REGION Network 28: pomocniczy bit ustawiania napędu dodatkowego nr2 / pomocniczy bit ustawiania pompy dodatkoweo nr2
   // Reset znacznika po udanym załączeniu pompy dodatkowej
   // Reset w wypadku braku pompy
   RUNG wire#powerrail
      I_Contact( "AlwaysTRUE" )
      wire#w1
      Contact( "Is_extras_K2_P1" )
      Contact( "IsRunNetwork_P1" )
      wire#w2
      R_Coil( #set_Motor3 )
   END_RUNG
   RUNG wire#w1
      Contact( "Is_extras_K2_P2" )
      Contact( "IsRunNetwork_P2" )
   END_RUNG wire#w2
   RUNG wire#w1
      Contact( "Is_extras_K2_P3" )
      Contact( "IsRunNetwork_P3" )
   END_RUNG wire#w2
   RUNG wire#w1
      Contact( "Is_extras_K2_P4" )
      Contact( "IsRunNetwork_P4" )
   END_RUNG wire#w2
   RUNG wire#w1
      Contact( "Reset_Motor3Alarm" )
   END_RUNG wire#w2
   RUNG wire#w1
      I_Contact( "IsModeAut" )
   END_RUNG wire#w2
   // the same network as SCL:
   IF NOT "AlwaysTRUE" AND (("Is_extras_K2_P1" AND "IsRunNetwork_P1") OR ("Is_extras_K2_P2" AND "IsRunNetwork_P2") OR ("Is_extras_K2_P3" AND "IsRunNetwork_P3") OR ("Is_extras_K2_P4" AND "IsRunNetwork_P4") OR "Reset_Motor3Alarm" OR NOT "IsModeAut") THEN
       #set_Motor3 := FALSE;
   END_IF;
END_REGION

REGION Network 29: pomocniczy bit ustawiania napędu dodatkowego nr2 / pomocniczy bit ustawiania pompy dodatkowe nr3
   // Reset znacznika po udanym załączeniu pompy dodatkowej
   // Reset w wypadku braku pompy
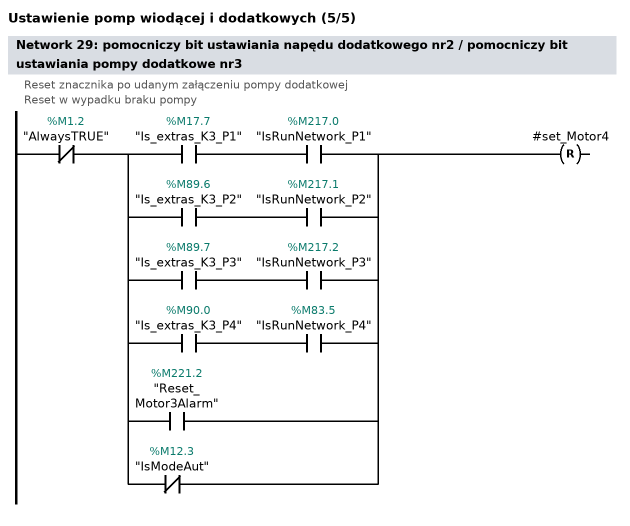
   RUNG wire#powerrail
      I_Contact( "AlwaysTRUE" )
      wire#w1
      Contact( "Is_extras_K3_P1" )
      Contact( "IsRunNetwork_P1" )
      wire#w2
      R_Coil( #set_Motor4 )
   END_RUNG
   RUNG wire#w1
      Contact( "Is_extras_K3_P2" )
      Contact( "IsRunNetwork_P2" )
   END_RUNG wire#w2
   RUNG wire#w1
      Contact( "Is_extras_K3_P3" )
      Contact( "IsRunNetwork_P3" )
   END_RUNG wire#w2
   RUNG wire#w1
      Contact( "Is_extras_K3_P4" )
      Contact( "IsRunNetwork_P4" )
   END_RUNG wire#w2
   RUNG wire#w1
      Contact( "Reset_Motor3Alarm" )
   END_RUNG wire#w2
   RUNG wire#w1
      I_Contact( "IsModeAut" )
   END_RUNG wire#w2
   // the same network as SCL:
   IF NOT "AlwaysTRUE" AND (("Is_extras_K3_P1" AND "IsRunNetwork_P1") OR ("Is_extras_K3_P2" AND "IsRunNetwork_P2") OR ("Is_extras_K3_P3" AND "IsRunNetwork_P3") OR ("Is_extras_K3_P4" AND "IsRunNetwork_P4") OR "Reset_Motor3Alarm" OR NOT "IsModeAut") THEN
       #set_Motor4 := FALSE;
   END_IF;
END_REGION
END_FUNCTION_BLOCK

FUNCTION_BLOCK "Sterowanie dołączeniem falownika"   // FB8, LAD
TITLE = Sterowanie dołączaniem styczników falownika
{ S7_Optimized_Access := 'TRUE' }
AUTHOR : rtecmer
VERSION : 0.1
// Sterowa stycznikiem pracy z falownika.
// Funkcja FB8 komutuje załaczenie stycznika FALOWNIK dla konkretnego napędu. Napędem sterowanym jest zawsze napęd przypisany do MC (czyli IsReady_MC to jest gotowość napędu sterowaniego) Na wejścia oznaczone wyróżnikiem MC podlączamy sygnały tej samej dmuchawy, której stycznikiem będziemy sterować poprzez wtjście setSUPV_FM
//  
// Sterowanie stycznikiem . Ustawianie znaczników setCMD_FM i setSUPV_FM które przekazywane są do funkcji FC3/FC1 DRV01 driver napędów. Następnie przekazywane jest do warstwy Hawtware/ OUT gdzie ustawiane jest wyjście sterownika
// stored: AutoNumber true, IsIECCheckEnabled false, IsRetainMemResEnabled false, MemoryReserve 500, SetENOAutomatically false, UDAEnableTagReadback false
   VAR_INPUT
      Is_up_Hz : Bool;
      Set_HWork_M : Bool;   // Znacznik ustawienia pracy od licznika
      setPID_Pompy : Bool;   // Znacznik załączenie, regulacji falownika
      IsRunInverter_MA : Bool;   // Potwierdzenie pracy z falownika kompresor dodatkowy 1
      IsRunNetwork_MA : Bool;   // Potwierdzenie praca z sieć dodatkowego
      IsRunInverter_MB : Bool;   // Potwierdzenie pracy z falownika kompresor dodatkowy 2
      IsRunNetwork_MB : Bool;   // Potwierdzenie praca z sieć dodatkowego
      IsRunNetwork_MC : Bool;   // Potwierdzenie pracy z sieci
      IsRunInverter_MC : Bool;   // Potwierdzenie pracy z falownika
      IsRunNetwork_MD : Bool;   // Potwierdzenie pracy z sieci
      IsRunInverter_MD : Bool;   // Potwierdzenie pracy z falownika
      FC2_Set_50H : Bool;   // Znacznik osiągnięcia czasu dla 50Hz
      IsRunInverter1 : Bool;   // Potwierdzenie pracy falownika / Potwierdzenie pracy falownika kompresorów M7M8M9
      AlwaysTRUE : Bool;
      IsReady_MA : Bool;   // Znacznik gotowości
      IsReady_MB : Bool;   // Znacznik gotowości
      IsReady_MC : Bool;   // Znacznik gotowości
      IsReady_MD : Bool;   // Znacznik gotowości
      IsModeAut : Bool;   // Znacznik trybu automat
      FB9_Set_Motor2 : Bool;   // Polecenie dostawienia dodatkowej nr1
      FB9_Set_Motor3 : Bool;   // Polecenie dostawienia dodatkowej nr2
      FB9_Set_Motor4 : Bool;   // Polecenie dostawienia dodatkowej nr3
      IsReady_Inverter : Bool;   // Gotowość falownika
      ResWorkInverter_to_MaxTime : Bool;   // Bit kasowania pracy falownika od maxymalnej ciągłej pracy
   END_VAR
   VAR_OUTPUT
      setSUPV_FM : Bool;   // Znacznik polecenia startu z falownika
   END_VAR
   VAR_IN_OUT
      setCMD_FM : Bool;   // Znacznik sterowania w trybie falownik
      Timer_OFF_Inverter_M : TOF_TIME;   // Timer na blokowanie po odłączeniu stycznika falownika
      Timer_Start_Inver_M : TON_TIME;   // Timer opóźnienia załaczenia stycznika pracy z falownika
      Timer_Set50Hz_Off_Inver_M : TON_TIME;   // Timer opóźnieniawyłączeniea falownika
      Mem_Res_setCMD_MC : Bool;   // pamięć zbocza załączenia timera blokowania stycznika falowni
   END_VAR
   VAR
      Network_50Hz : Bool;   // Znacznik 50 Hz podtrzymanie przełączenia na sieć
   END_VAR
   VAR_TEMP
      IsDrive_Optimum : Bool;   // Znacznik optymalnej ilości napędów. Jeśli False to nie przełaczaj Falowni/Sieć
      CMD_OFF_inverter : Bool;   // Wyłączenie falownika od 50Hz i dodatkowa / Wyłączenie falownika od 50Hz i udtawiona dodatkowa
      tmpOFF_inverter : Bool;
   END_VAR
   VAR_TEMP   // added for the SCL form of the ladder/FBD networks
      _w1 : Bool;
      _w2 : Bool;
   END_VAR
BEGIN

REGION Network 1: Control status motors / Kontrola statusu napędu
   // // Dostępna  jedna dmuchawa gdy wartość 1, 2, 4
   // // Dostępne dwie dmuchawy gdy wartość 6, 5, 3 
   // // Dostępne trzy dmuchawy gdy wartość 7
END_REGION

REGION Network 2: Histereza na dołączenie stycznika falownika
   // Sterowanie dołączeniem stycznika pracy z falownika
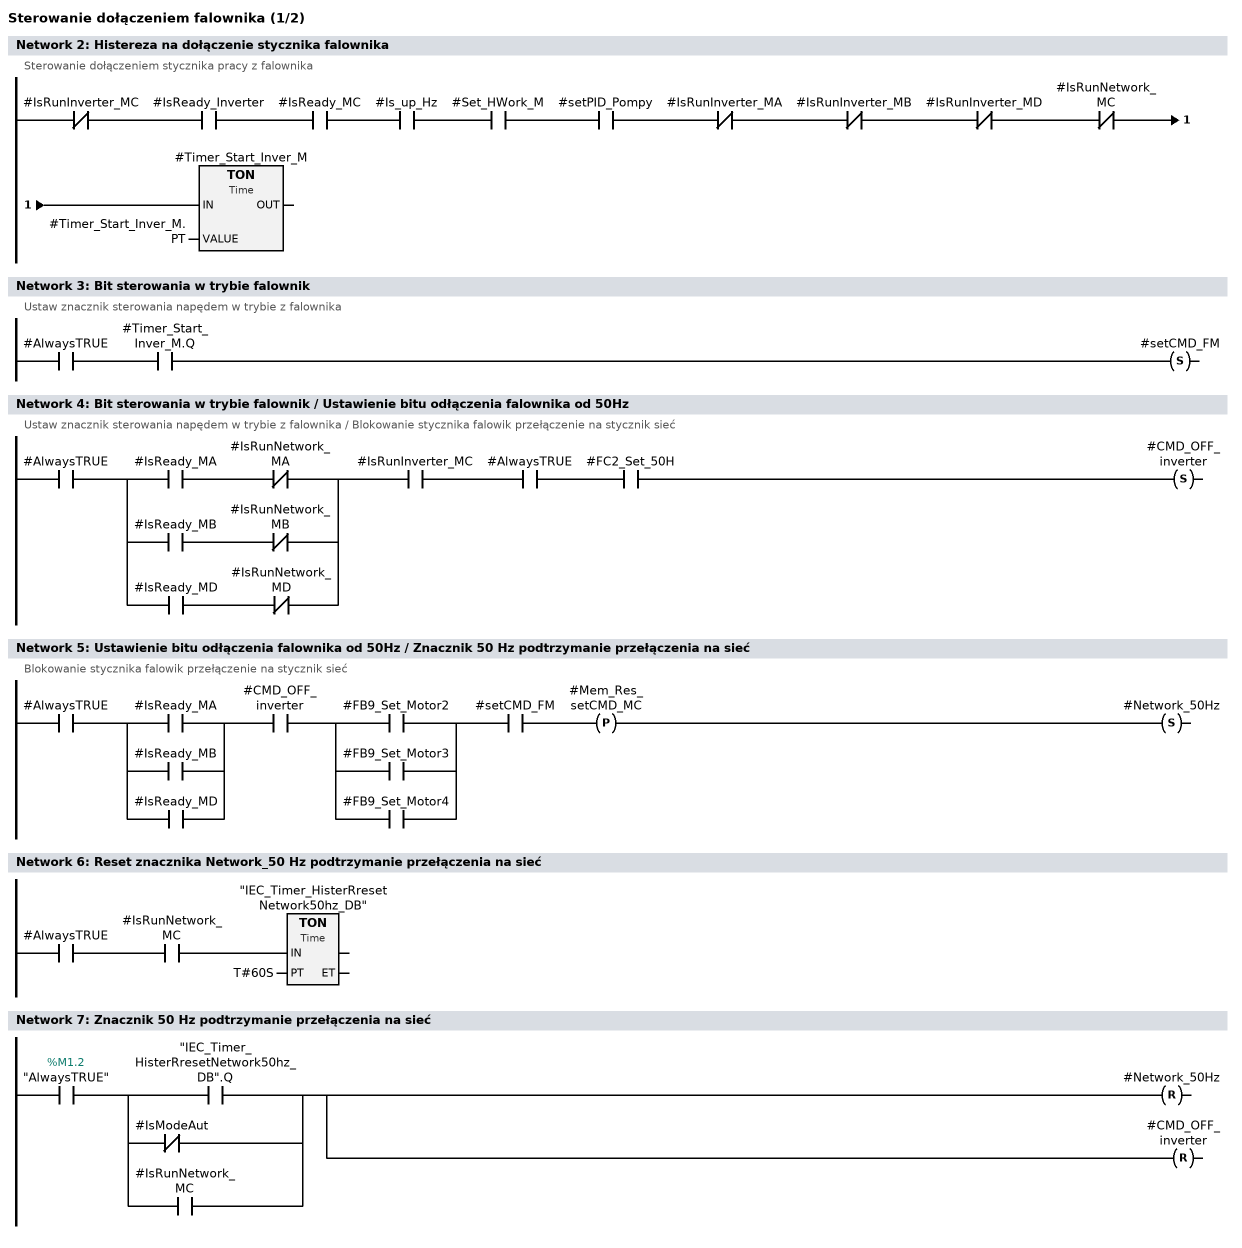
   #Timer_Start_Inver_M(IN := NOT #IsRunInverter_MC AND #IsReady_Inverter AND #IsReady_MC AND #Is_up_Hz AND #Set_HWork_M AND #setPID_Pompy AND NOT #IsRunInverter_MA AND NOT #IsRunInverter_MB AND NOT #IsRunInverter_MD AND NOT #IsRunNetwork_MC, PT := #Timer_Start_Inver_M.PT);   // TON coil
END_REGION

REGION Network 3: Bit sterowania w trybie falownik
   // Ustaw znacznik sterowania napędem w trybie z falownika
   RUNG wire#powerrail
      Contact( #AlwaysTRUE )
      Contact( #Timer_Start_Inver_M.Q )
      S_Coil( #setCMD_FM )
   END_RUNG
   // the same network as SCL:
   IF #AlwaysTRUE AND #Timer_Start_Inver_M.Q THEN #setCMD_FM := TRUE; END_IF;
END_REGION

REGION Network 4: Bit sterowania w trybie falownik / Ustawienie bitu odłączenia falownika od 50Hz
   // Ustaw znacznik sterowania napędem w trybie z falownika / Blokowanie stycznika falowik przełączenie na stycznik sieć
   RUNG wire#powerrail
      Contact( #AlwaysTRUE )
      wire#w1
      Contact( #IsReady_MA )
      I_Contact( #IsRunNetwork_MA )
      wire#w2
      Contact( #IsRunInverter_MC )
      Contact( #AlwaysTRUE )
      Contact( #FC2_Set_50H )
      S_Coil( #CMD_OFF_inverter )
   END_RUNG
   RUNG wire#w1
      Contact( #IsReady_MB )
      I_Contact( #IsRunNetwork_MB )
   END_RUNG wire#w2
   RUNG wire#w1
      Contact( #IsReady_MD )
      I_Contact( #IsRunNetwork_MD )
   END_RUNG wire#w2
   // the same network as SCL:
   IF #AlwaysTRUE AND ((#IsReady_MA AND NOT #IsRunNetwork_MA) OR (#IsReady_MB AND NOT #IsRunNetwork_MB) OR (#IsReady_MD AND NOT #IsRunNetwork_MD)) AND #IsRunInverter_MC AND #AlwaysTRUE AND #FC2_Set_50H THEN
       #CMD_OFF_inverter := TRUE;
   END_IF;
END_REGION

REGION Network 5: Ustawienie bitu odłączenia falownika od 50Hz / Znacznik 50 Hz podtrzymanie przełączenia na sieć
   // Blokowanie stycznika falowik przełączenie na stycznik sieć
   RUNG wire#powerrail
      Contact( #AlwaysTRUE )
      wire#w1
      Contact( #IsReady_MA )
      wire#w2
      Contact( #CMD_OFF_inverter )
      wire#w3
      Contact( #FB9_Set_Motor2 )
      wire#w4
      Contact( #setCMD_FM )
      P_Trig( #Mem_Res_setCMD_MC )
      S_Coil( #Network_50Hz )
   END_RUNG
   RUNG wire#w1
      Contact( #IsReady_MB )
   END_RUNG wire#w2
   RUNG wire#w1
      Contact( #IsReady_MD )
   END_RUNG wire#w2
   RUNG wire#w3
      Contact( #FB9_Set_Motor3 )
   END_RUNG wire#w4
   RUNG wire#w3
      Contact( #FB9_Set_Motor4 )
   END_RUNG wire#w4
   // the same network as SCL:
   #_w1 := #AlwaysTRUE AND (#IsReady_MA OR #IsReady_MB OR #IsReady_MD) AND #CMD_OFF_inverter AND (#FB9_Set_Motor2 OR #FB9_Set_Motor3 OR #FB9_Set_Motor4) AND #setCMD_FM;
   #_w2 := #_w1 AND NOT #Mem_Res_setCMD_MC;   // rising edge
   #Mem_Res_setCMD_MC := #_w1;
   IF #_w2 THEN #Network_50Hz := TRUE; END_IF;
END_REGION

REGION Network 6: Reset znacznika Network_50 Hz podtrzymanie przełączenia na sieć
   RUNG wire#powerrail
      Contact( #AlwaysTRUE )
      Contact( #IsRunNetwork_MC )
      { S7_Templates := "time_type := Time" } "IEC_Timer_HisterRresetNetwork50hz_DB".TON(pt := T#60S, et =>)
   END_RUNG
   // the same network as SCL:
   "IEC_Timer_HisterRresetNetwork50hz_DB".TON(IN := #AlwaysTRUE AND #IsRunNetwork_MC, PT := T#60S);
END_REGION

REGION Network 7: Znacznik 50 Hz podtrzymanie przełączenia na sieć
   RUNG wire#powerrail
      Contact( "AlwaysTRUE" )
      wire#w1
      Contact( "IEC_Timer_HisterRresetNetwork50hz_DB".Q )
      wire#w2
      R_Coil( #Network_50Hz )
   END_RUNG
   RUNG wire#w1
      I_Contact( #IsModeAut )
   END_RUNG wire#w2
   RUNG wire#w1
      Contact( #IsRunNetwork_MC )
   END_RUNG wire#w2
   RUNG wire#w2
      R_Coil( #CMD_OFF_inverter )
   END_RUNG
   // the same network as SCL:
   IF "AlwaysTRUE" AND ("IEC_Timer_HisterRresetNetwork50hz_DB".Q OR NOT #IsModeAut OR #IsRunNetwork_MC) THEN
       #Network_50Hz := FALSE;
       #CMD_OFF_inverter := FALSE;
   END_IF;
END_REGION

REGION Network 8: Timer blokowania po odłączenieu stycznika falownik
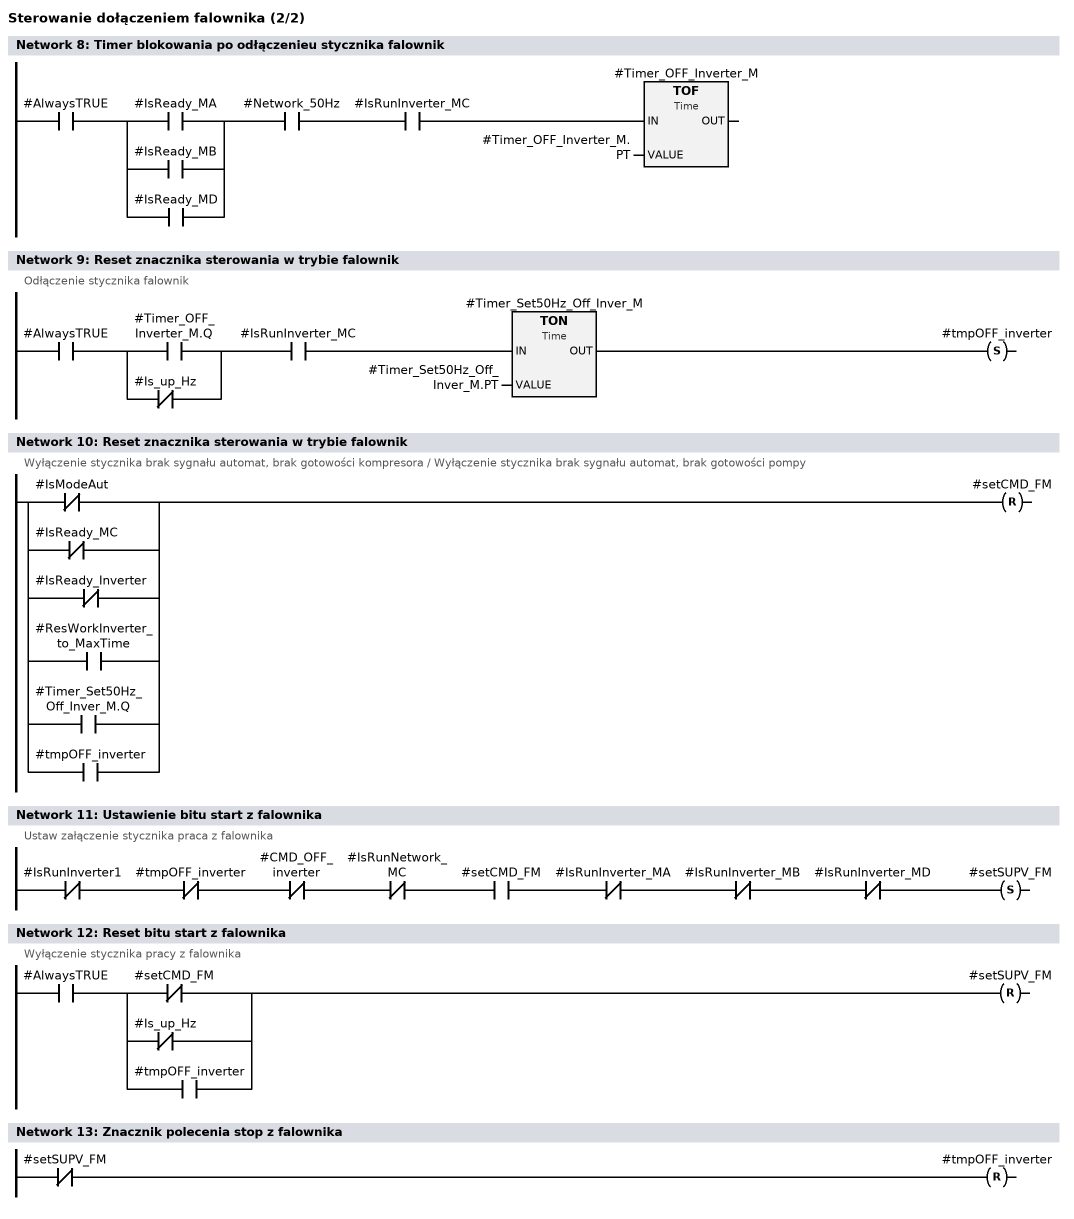
   #Timer_OFF_Inverter_M(IN := #AlwaysTRUE AND (#IsReady_MA OR #IsReady_MB OR #IsReady_MD) AND #Network_50Hz AND #IsRunInverter_MC, PT := #Timer_OFF_Inverter_M.PT);   // TOF coil
END_REGION

REGION Network 9: Reset znacznika sterowania w trybie falownik
   // Odłączenie stycznika falownik
   #_w1 := #AlwaysTRUE AND (#Timer_OFF_Inverter_M.Q OR NOT #Is_up_Hz) AND #IsRunInverter_MC;
   #Timer_Set50Hz_Off_Inver_M(IN := #_w1, PT := #Timer_Set50Hz_Off_Inver_M.PT);   // TON coil
   IF #_w1 THEN #tmpOFF_inverter := TRUE; END_IF;
END_REGION

REGION Network 10: Reset znacznika sterowania w trybie falownik
   // Wyłączenie stycznika brak sygnału automat, brak gotowości kompresora / Wyłączenie stycznika brak sygnału automat, brak gotowości pompy
   RUNG wire#powerrail
      I_Contact( #IsModeAut )
      wire#w1
      R_Coil( #setCMD_FM )
   END_RUNG
   RUNG wire#powerrail
      I_Contact( #IsReady_MC )
   END_RUNG wire#w1
   RUNG wire#powerrail
      I_Contact( #IsReady_Inverter )
   END_RUNG wire#w1
   RUNG wire#powerrail
      Contact( #ResWorkInverter_to_MaxTime )
   END_RUNG wire#w1
   RUNG wire#powerrail
      Contact( #Timer_Set50Hz_Off_Inver_M.Q )
   END_RUNG wire#w1
   RUNG wire#powerrail
      Contact( #tmpOFF_inverter )
   END_RUNG wire#w1
   // the same network as SCL:
   IF NOT #IsModeAut OR NOT #IsReady_MC OR NOT #IsReady_Inverter OR #ResWorkInverter_to_MaxTime OR #Timer_Set50Hz_Off_Inver_M.Q OR #tmpOFF_inverter THEN
       #setCMD_FM := FALSE;
   END_IF;
END_REGION

REGION Network 11: Ustawienie bitu start z falownika
   // Ustaw załączenie stycznika praca z falownika
   RUNG wire#powerrail
      I_Contact( #IsRunInverter1 )
      I_Contact( #tmpOFF_inverter )
      I_Contact( #CMD_OFF_inverter )
      I_Contact( #IsRunNetwork_MC )
      Contact( #setCMD_FM )
      I_Contact( #IsRunInverter_MA )
      I_Contact( #IsRunInverter_MB )
      I_Contact( #IsRunInverter_MD )
      S_Coil( #setSUPV_FM )
   END_RUNG
   // the same network as SCL:
   IF NOT #IsRunInverter1 AND NOT #tmpOFF_inverter AND NOT #CMD_OFF_inverter AND NOT #IsRunNetwork_MC AND #setCMD_FM AND NOT #IsRunInverter_MA AND NOT #IsRunInverter_MB AND NOT #IsRunInverter_MD THEN
       #setSUPV_FM := TRUE;
   END_IF;
END_REGION

REGION Network 12: Reset bitu start z falownika
   // Wyłączenie stycznika pracy z falownika
   RUNG wire#powerrail
      Contact( #AlwaysTRUE )
      wire#w1
      I_Contact( #setCMD_FM )
      wire#w2
      R_Coil( #setSUPV_FM )
   END_RUNG
   RUNG wire#w1
      I_Contact( #Is_up_Hz )
   END_RUNG wire#w2
   RUNG wire#w1
      Contact( #tmpOFF_inverter )
   END_RUNG wire#w2
   // the same network as SCL:
   IF #AlwaysTRUE AND (NOT #setCMD_FM OR NOT #Is_up_Hz OR #tmpOFF_inverter) THEN
       #setSUPV_FM := FALSE;
   END_IF;
END_REGION

REGION Network 13: Znacznik polecenia stop z falownika
   RUNG wire#powerrail
      I_Contact( #setSUPV_FM )
      R_Coil( #tmpOFF_inverter )
   END_RUNG
   // the same network as SCL:
   IF NOT #setSUPV_FM THEN #tmpOFF_inverter := FALSE; END_IF;
END_REGION
END_FUNCTION_BLOCK

FUNCTION "Korekta Tryb Pracy" : Void   // FC34, LAD
TITLE = potrzymanie trybu
{ S7_Optimized_Access := 'TRUE' }
AUTHOR : rtecmer
VERSION : 0.1
// z powodu P1 dodanyblok potzymujący tryb pracy napędów podczas przełączania falowni / siec
// stored: AutoNumber true, IsIECCheckEnabled false, SetENOAutomatically false, UDAEnableTagReadback false
   VAR_TEMP   // added for the SCL form of the ladder/FBD networks
      _w1 : Bool;
   END_VAR
BEGIN

REGION Network 2: Ustawienie pracy [Automat]
   // Ustawienie bitu [Automat] przełacznikiem trybu pracy
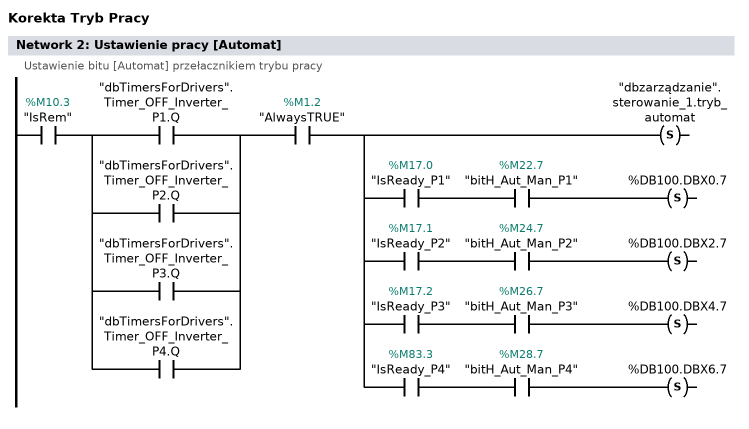
   RUNG wire#powerrail
      Contact( "IsRem" )
      wire#w1
      Contact( "dbTimersForDrivers".Timer_OFF_Inverter_P1.Q )
      wire#w2
      Contact( "AlwaysTRUE" )
      wire#w3
      S_Coil( "dbzarządzanie".sterowanie_1.tryb_automat )
   END_RUNG
   RUNG wire#w1
      Contact( "dbTimersForDrivers".Timer_OFF_Inverter_P2.Q )
   END_RUNG wire#w2
   RUNG wire#w1
      Contact( "dbTimersForDrivers".Timer_OFF_Inverter_P3.Q )
   END_RUNG wire#w2
   RUNG wire#w1
      Contact( "dbTimersForDrivers".Timer_OFF_Inverter_P4.Q )
   END_RUNG wire#w2
   RUNG wire#w3
      Contact( "IsReady_P1" )
      Contact( "bitH_Aut_Man_P1" )
      S_Coil( %DB100.DBX0.7 )
   END_RUNG
   RUNG wire#w3
      Contact( "IsReady_P2" )
      Contact( "bitH_Aut_Man_P2" )
      S_Coil( %DB100.DBX2.7 )
   END_RUNG
   RUNG wire#w3
      Contact( "IsReady_P3" )
      Contact( "bitH_Aut_Man_P3" )
      S_Coil( %DB100.DBX4.7 )
   END_RUNG
   RUNG wire#w3
      Contact( "IsReady_P4" )
      Contact( "bitH_Aut_Man_P4" )
      S_Coil( %DB100.DBX6.7 )
   END_RUNG
   // the same network as SCL:
   #_w1 := "IsRem" AND ("dbTimersForDrivers".Timer_OFF_Inverter_P1.Q OR "dbTimersForDrivers".Timer_OFF_Inverter_P2.Q OR "dbTimersForDrivers".Timer_OFF_Inverter_P3.Q OR "dbTimersForDrivers".Timer_OFF_Inverter_P4.Q) AND "AlwaysTRUE";
   IF #_w1 THEN "dbzarządzanie".sterowanie_1.tryb_automat := TRUE; END_IF;
   IF #_w1 AND "IsReady_P1" AND "bitH_Aut_Man_P1" THEN %DB100.DBX0.7 := TRUE; END_IF;
   IF #_w1 AND "IsReady_P2" AND "bitH_Aut_Man_P2" THEN %DB100.DBX2.7 := TRUE; END_IF;
   IF #_w1 AND "IsReady_P3" AND "bitH_Aut_Man_P3" THEN %DB100.DBX4.7 := TRUE; END_IF;
   IF #_w1 AND "IsReady_P4" AND "bitH_Aut_Man_P4" THEN %DB100.DBX6.7 := TRUE; END_IF;
END_REGION
END_FUNCTION

FUNCTION_BLOCK "Sterowanie falownikiem"   // FB11, LAD
TITLE = Control of Inverters
{ S7_Optimized_Access := 'TRUE' }
AUTHOR : rtecmer
VERSION : 0.1
// Sterowanie przekaćnikiem załączającym falownik do pracy
// stored: AutoNumber true, IsIECCheckEnabled false, IsRetainMemResEnabled false, MemoryReserve 500, SetENOAutomatically false, UDAEnableTagReadback false
   VAR_INPUT
      IsModeAut : Bool;   // Znacznik tryb automat dla pomp
      AlwaysTRUE : Bool;
      Set_HWork_P1 : Bool;   // Znacznik ustawienia pracy od licznika pracy
      Set_HWork_P2 : Bool;   // Znacznik ustawienia pracy od licznika pracy
      Set_HWork_P3 : Bool;   // Znacznik ustawienia pracy od licznika pracy
      Set_HWork_P4 : Bool;
      setPID_Pomp : Bool;   // Znacznik załączenie, regulacji falownika
      Is_loading_K3 : Bool;   // Znacznik pompy wiodącej
      IsRunInverter_P4 : Bool;
      IsRunInverter_P3 : Bool;   // Potwierdzenie załączenie stycznika falownik pompy
      IsRunInverter_P2 : Bool;   // Potwierdzenie załączenie stycznika falownik pompy
      IsRunInverter_P1 : Bool;   // Potwierdzenie załączenie stycznika falownik pompy
      Bit_Aut_P1 : Bool;   // Bit tryb prac automat
      Bit_Aut_P2 : Bool;   // Bit tryb prac automat
      Bit_Aut_P3 : Bool;   // Bit tryb prac automat
      Bit_Aut_P4 : Bool;
      IsRunNetwork_P1 : Bool;   // Potwierdzenie załączenie stycznika sieć
      IsRunNetwork_P2 : Bool := false;   // Potwierdzenie załączenie stycznika sieć
      IsRunNetwork_P3 : Bool := false;   // Potwierdzenie załączenie stycznika sieć
      IsRunNetwork_P4 : Bool;
   END_VAR
   VAR_OUTPUT
      CMD_start_stop_inverter : Bool;   // Przekaźnik sterowania załączaniem falownika
   END_VAR
   VAR
      Res_upHz : Bool;   // Reset znacznika up_Hz wyłaczenie dodatkowe
   END_VAR
BEGIN

REGION Network 1: Reset bitu pomocniczego ustalenia przyrostu Hz
   // Kasowanie podczas rozruchu po restarcie
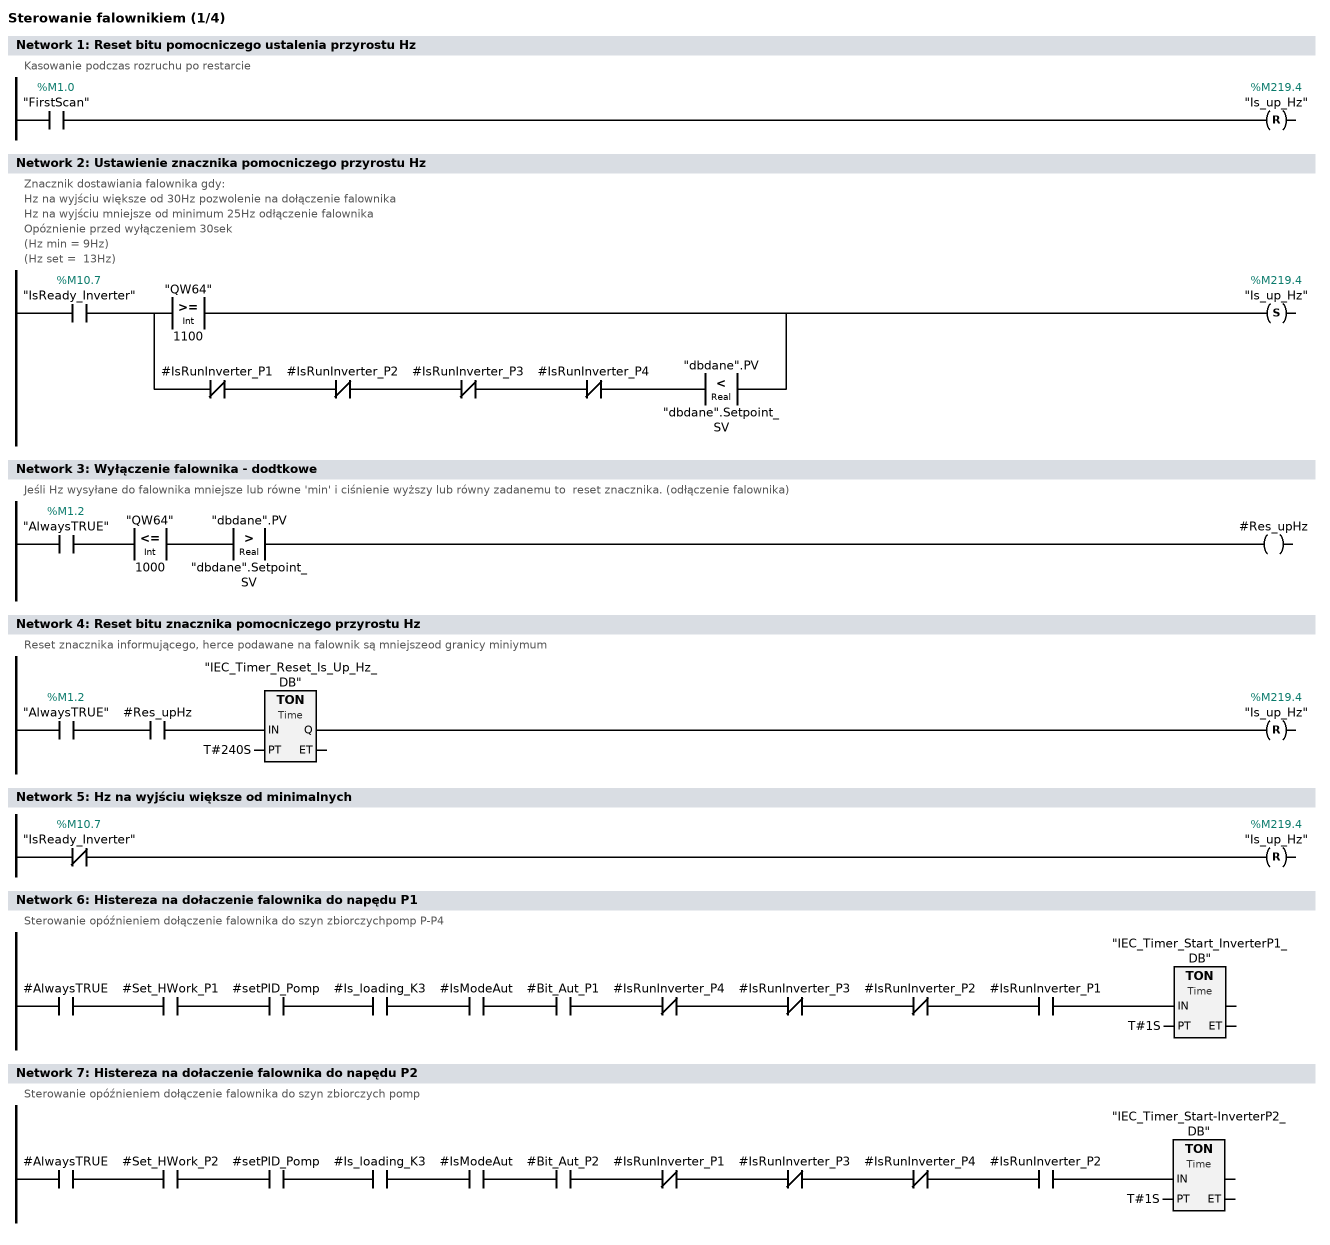
   RUNG wire#powerrail
      Contact( "FirstScan" )
      R_Coil( "Is_up_Hz" )
   END_RUNG
   // the same network as SCL:
   IF "FirstScan" THEN "Is_up_Hz" := FALSE; END_IF;
END_REGION

REGION Network 2: Ustawienie znacznika pomocniczego przyrostu Hz
   // Znacznik dostawiania falownika gdy:
   // Hz na wyjściu większe od 30Hz pozwolenie na dołączenie falownika
   // Hz na wyjściu mniejsze od minimum 25Hz odłączenie falownika
   // Opóznienie przed wyłączeniem 30sek
   // (Hz min = 9Hz)
   // (Hz set =  13Hz)
   RUNG wire#powerrail
      Contact( "IsReady_Inverter" )
      wire#w1
      { S7_Templates := "SrcType := Int" } GE_Contact(in1 := "QW64", in2 := 1100)
      wire#w2
      S_Coil( "Is_up_Hz" )
   END_RUNG
   RUNG wire#w1
      I_Contact( #IsRunInverter_P1 )
      I_Contact( #IsRunInverter_P2 )
      I_Contact( #IsRunInverter_P3 )
      I_Contact( #IsRunInverter_P4 )
      { S7_Templates := "SrcType := Real" } LT_Contact(in1 := "dbdane".PV, in2 := "dbdane".Setpoint_SV)
   END_RUNG wire#w2
   // the same network as SCL:
   IF "IsReady_Inverter" AND (("QW64" >= 1100) OR (NOT #IsRunInverter_P1 AND NOT #IsRunInverter_P2 AND NOT #IsRunInverter_P3 AND NOT #IsRunInverter_P4 AND ("dbdane".PV < "dbdane".Setpoint_SV))) THEN
       "Is_up_Hz" := TRUE;
   END_IF;
END_REGION

REGION Network 3: Wyłączenie falownika - dodtkowe
   // Jeśli Hz wysyłane do falownika mniejsze lub równe 'min' i ciśnienie wyższy lub równy zadanemu to  reset znacznika. (odłączenie falownika)
   RUNG wire#powerrail
      Contact( "AlwaysTRUE" )
      { S7_Templates := "SrcType := Int" } LE_Contact(in1 := "QW64", in2 := 1000)
      { S7_Templates := "SrcType := Real" } GT_Contact(in1 := "dbdane".PV, in2 := "dbdane".Setpoint_SV)
      Coil( #Res_upHz )
   END_RUNG
   // the same network as SCL:
   #Res_upHz := "AlwaysTRUE" AND ("QW64" <= 1000) AND ("dbdane".PV > "dbdane".Setpoint_SV);
END_REGION

REGION Network 4: Reset bitu znacznika pomocniczego przyrostu Hz
   // Reset znacznika informującego, herce podawane na falownik są mniejszeod granicy miniymum
   RUNG wire#powerrail
      Contact( "AlwaysTRUE" )
      Contact( #Res_upHz )
      { S7_Templates := "time_type := Time" } "IEC_Timer_Reset_Is_Up_Hz_DB".TON(pt := T#240S, et =>)
      R_Coil( "Is_up_Hz" )
   END_RUNG
   // the same network as SCL:
   "IEC_Timer_Reset_Is_Up_Hz_DB".TON(IN := "AlwaysTRUE" AND #Res_upHz, PT := T#240S);
   IF "IEC_Timer_Reset_Is_Up_Hz_DB".Q THEN "Is_up_Hz" := FALSE; END_IF;
END_REGION

REGION Network 5: Hz na wyjściu większe od minimalnych
   RUNG wire#powerrail
      I_Contact( "IsReady_Inverter" )
      R_Coil( "Is_up_Hz" )
   END_RUNG
   // the same network as SCL:
   IF NOT "IsReady_Inverter" THEN "Is_up_Hz" := FALSE; END_IF;
END_REGION

REGION Network 6: Histereza na dołaczenie falownika do napędu P1
   // Sterowanie opóźnieniem dołączenie falownika do szyn zbiorczychpomp P-P4
   RUNG wire#powerrail
      Contact( #AlwaysTRUE )
      Contact( #Set_HWork_P1 )
      Contact( #setPID_Pomp )
      Contact( #Is_loading_K3 )
      Contact( #IsModeAut )
      Contact( #Bit_Aut_P1 )
      I_Contact( #IsRunInverter_P4 )
      I_Contact( #IsRunInverter_P3 )
      I_Contact( #IsRunInverter_P2 )
      Contact( #IsRunInverter_P1 )
      { S7_Templates := "time_type := Time" } "IEC_Timer_Start_InverterP1_DB".TON(pt := T#1S, et =>)
   END_RUNG
   // the same network as SCL:
   "IEC_Timer_Start_InverterP1_DB".TON(IN := #AlwaysTRUE AND #Set_HWork_P1 AND #setPID_Pomp AND #Is_loading_K3 AND #IsModeAut AND #Bit_Aut_P1 AND NOT #IsRunInverter_P4 AND NOT #IsRunInverter_P3 AND NOT #IsRunInverter_P2 AND #IsRunInverter_P1,
                           PT := T#1S);
END_REGION

REGION Network 7: Histereza na dołaczenie falownika do napędu P2
   // Sterowanie opóźnieniem dołączenie falownika do szyn zbiorczych pomp
   RUNG wire#powerrail
      Contact( #AlwaysTRUE )
      Contact( #Set_HWork_P2 )
      Contact( #setPID_Pomp )
      Contact( #Is_loading_K3 )
      Contact( #IsModeAut )
      Contact( #Bit_Aut_P2 )
      I_Contact( #IsRunInverter_P1 )
      I_Contact( #IsRunInverter_P3 )
      I_Contact( #IsRunInverter_P4 )
      Contact( #IsRunInverter_P2 )
      { S7_Templates := "time_type := Time" } "IEC_Timer_Start-InverterP2_DB".TON(pt := T#1S, et =>)
   END_RUNG
   // the same network as SCL:
   "IEC_Timer_Start-InverterP2_DB".TON(IN := #AlwaysTRUE AND #Set_HWork_P2 AND #setPID_Pomp AND #Is_loading_K3 AND #IsModeAut AND #Bit_Aut_P2 AND NOT #IsRunInverter_P1 AND NOT #IsRunInverter_P3 AND NOT #IsRunInverter_P4 AND #IsRunInverter_P2,
                           PT := T#1S);
END_REGION

REGION Network 8: Histereza na dołaczenie falownika do napędu P3
   // Sterowanie opóźnieniem dołączenie falownika do szyn zbiorczych kompresorów
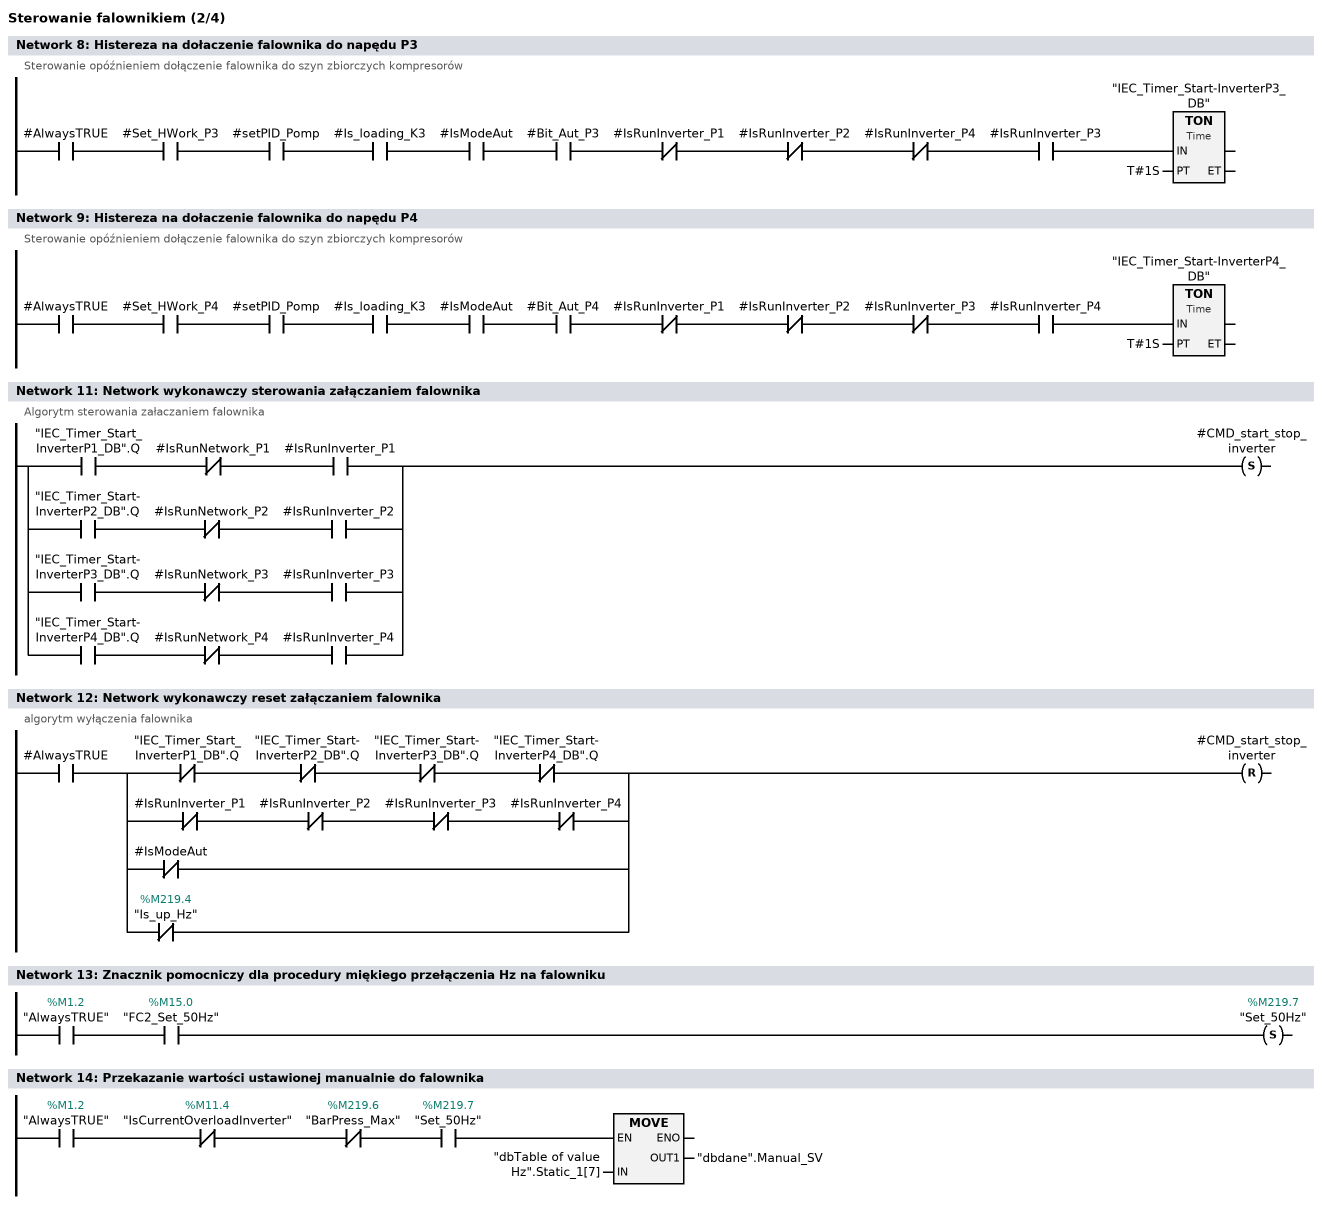
   RUNG wire#powerrail
      Contact( #AlwaysTRUE )
      Contact( #Set_HWork_P3 )
      Contact( #setPID_Pomp )
      Contact( #Is_loading_K3 )
      Contact( #IsModeAut )
      Contact( #Bit_Aut_P3 )
      I_Contact( #IsRunInverter_P1 )
      I_Contact( #IsRunInverter_P2 )
      I_Contact( #IsRunInverter_P4 )
      Contact( #IsRunInverter_P3 )
      { S7_Templates := "time_type := Time" } "IEC_Timer_Start-InverterP3_DB".TON(pt := T#1S, et =>)
   END_RUNG
   // the same network as SCL:
   "IEC_Timer_Start-InverterP3_DB".TON(IN := #AlwaysTRUE AND #Set_HWork_P3 AND #setPID_Pomp AND #Is_loading_K3 AND #IsModeAut AND #Bit_Aut_P3 AND NOT #IsRunInverter_P1 AND NOT #IsRunInverter_P2 AND NOT #IsRunInverter_P4 AND #IsRunInverter_P3,
                           PT := T#1S);
END_REGION

REGION Network 9: Histereza na dołaczenie falownika do napędu P4
   // Sterowanie opóźnieniem dołączenie falownika do szyn zbiorczych kompresorów
   RUNG wire#powerrail
      Contact( #AlwaysTRUE )
      Contact( #Set_HWork_P4 )
      Contact( #setPID_Pomp )
      Contact( #Is_loading_K3 )
      Contact( #IsModeAut )
      Contact( #Bit_Aut_P4 )
      I_Contact( #IsRunInverter_P1 )
      I_Contact( #IsRunInverter_P2 )
      I_Contact( #IsRunInverter_P3 )
      Contact( #IsRunInverter_P4 )
      { S7_Templates := "time_type := Time" } "IEC_Timer_Start-InverterP4_DB".TON(pt := T#1S, et =>)
   END_RUNG
   // the same network as SCL:
   "IEC_Timer_Start-InverterP4_DB".TON(IN := #AlwaysTRUE AND #Set_HWork_P4 AND #setPID_Pomp AND #Is_loading_K3 AND #IsModeAut AND #Bit_Aut_P4 AND NOT #IsRunInverter_P1 AND NOT #IsRunInverter_P2 AND NOT #IsRunInverter_P3 AND #IsRunInverter_P4,
                           PT := T#1S);
END_REGION

REGION Network 11: Network wykonawczy sterowania załączaniem falownika
   // Algorytm sterowania załaczaniem falownika
   RUNG wire#powerrail
      Contact( "IEC_Timer_Start_InverterP1_DB".Q )
      I_Contact( #IsRunNetwork_P1 )
      Contact( #IsRunInverter_P1 )
      wire#w1
      S_Coil( #CMD_start_stop_inverter )
   END_RUNG
   RUNG wire#powerrail
      Contact( "IEC_Timer_Start-InverterP2_DB".Q )
      I_Contact( #IsRunNetwork_P2 )
      Contact( #IsRunInverter_P2 )
   END_RUNG wire#w1
   RUNG wire#powerrail
      Contact( "IEC_Timer_Start-InverterP3_DB".Q )
      I_Contact( #IsRunNetwork_P3 )
      Contact( #IsRunInverter_P3 )
   END_RUNG wire#w1
   RUNG wire#powerrail
      Contact( "IEC_Timer_Start-InverterP4_DB".Q )
      I_Contact( #IsRunNetwork_P4 )
      Contact( #IsRunInverter_P4 )
   END_RUNG wire#w1
   // the same network as SCL:
   IF ("IEC_Timer_Start_InverterP1_DB".Q AND NOT #IsRunNetwork_P1 AND #IsRunInverter_P1) OR ("IEC_Timer_Start-InverterP2_DB".Q AND NOT #IsRunNetwork_P2 AND #IsRunInverter_P2) OR ("IEC_Timer_Start-InverterP3_DB".Q AND NOT #IsRunNetwork_P3 AND #IsRunInverter_P3) OR ("IEC_Timer_Start-InverterP4_DB".Q AND NOT #IsRunNetwork_P4 AND #IsRunInverter_P4) THEN
       #CMD_start_stop_inverter := TRUE;
   END_IF;
END_REGION

REGION Network 12: Network wykonawczy reset załączaniem falownika
   // algorytm wyłączenia falownika
   RUNG wire#powerrail
      Contact( #AlwaysTRUE )
      wire#w1
      I_Contact( "IEC_Timer_Start_InverterP1_DB".Q )
      I_Contact( "IEC_Timer_Start-InverterP2_DB".Q )
      I_Contact( "IEC_Timer_Start-InverterP3_DB".Q )
      I_Contact( "IEC_Timer_Start-InverterP4_DB".Q )
      wire#w2
      R_Coil( #CMD_start_stop_inverter )
   END_RUNG
   RUNG wire#w1
      I_Contact( #IsRunInverter_P1 )
      I_Contact( #IsRunInverter_P2 )
      I_Contact( #IsRunInverter_P3 )
      I_Contact( #IsRunInverter_P4 )
   END_RUNG wire#w2
   RUNG wire#w1
      I_Contact( #IsModeAut )
   END_RUNG wire#w2
   RUNG wire#w1
      I_Contact( "Is_up_Hz" )
   END_RUNG wire#w2
   // the same network as SCL:
   IF #AlwaysTRUE AND ((NOT "IEC_Timer_Start_InverterP1_DB".Q AND NOT "IEC_Timer_Start-InverterP2_DB".Q AND NOT "IEC_Timer_Start-InverterP3_DB".Q AND NOT "IEC_Timer_Start-InverterP4_DB".Q) OR (NOT #IsRunInverter_P1 AND NOT #IsRunInverter_P2 AND NOT #IsRunInverter_P3 AND NOT #IsRunInverter_P4) OR NOT #IsModeAut OR NOT "Is_up_Hz") THEN
       #CMD_start_stop_inverter := FALSE;
   END_IF;
END_REGION

REGION Network 13: Znacznik pomocniczy dla procedury miękiego przełączenia Hz na falowniku
   RUNG wire#powerrail
      Contact( "AlwaysTRUE" )
      Contact( "FC2_Set_50Hz" )
      S_Coil( "Set_50Hz" )
   END_RUNG
   // the same network as SCL:
   IF "AlwaysTRUE" AND "FC2_Set_50Hz" THEN "Set_50Hz" := TRUE; END_IF;
END_REGION

REGION Network 14: Przekazanie wartości ustawionej manualnie do falownika
   RUNG wire#powerrail
      Contact( "AlwaysTRUE" )
      I_Contact( "IsCurrentOverloadInverter" )
      I_Contact( "BarPress_Max" )
      Contact( "Set_50Hz" )
      Move(in := "dbTable of value Hz".Static_1[7], out1 => "dbdane".Manual_SV)
   END_RUNG
   // the same network as SCL:
   IF "AlwaysTRUE" AND NOT "IsCurrentOverloadInverter" AND NOT "BarPress_Max" AND "Set_50Hz" THEN
       "dbdane".Manual_SV := "dbTable of value Hz".Static_1[7];
   END_IF;
END_REGION

REGION Network 15: Przekazanie wartości ustawionej manualnie do falownika gdy awaria max ciśnienie
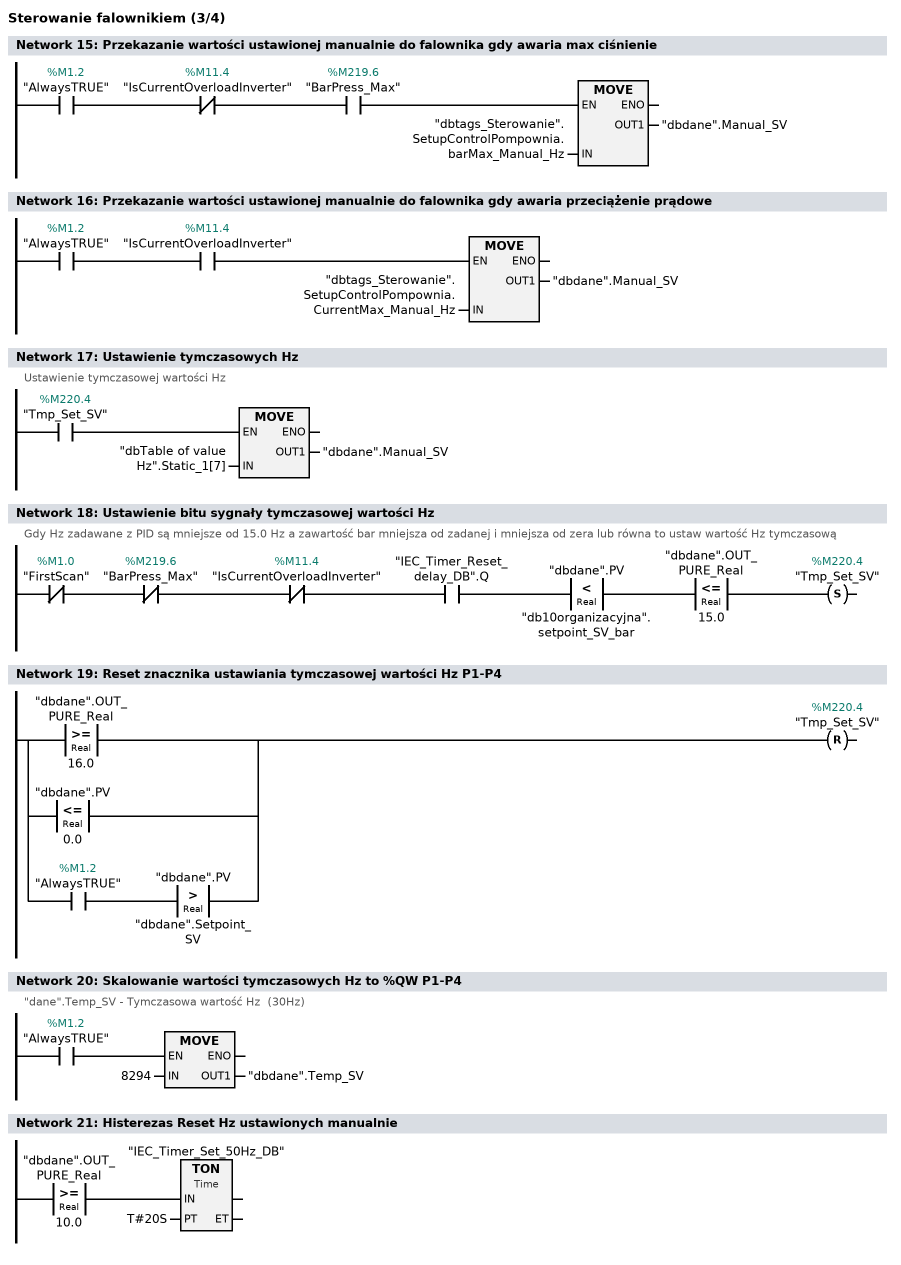
   RUNG wire#powerrail
      Contact( "AlwaysTRUE" )
      I_Contact( "IsCurrentOverloadInverter" )
      Contact( "BarPress_Max" )
      Move(in := "dbtags_Sterowanie".SetupControlPompownia.barMax_Manual_Hz, out1 => "dbdane".Manual_SV)
   END_RUNG
   // the same network as SCL:
   IF "AlwaysTRUE" AND NOT "IsCurrentOverloadInverter" AND "BarPress_Max" THEN
       "dbdane".Manual_SV := "dbtags_Sterowanie".SetupControlPompownia.barMax_Manual_Hz;
   END_IF;
END_REGION

REGION Network 16: Przekazanie wartości ustawionej manualnie do falownika gdy awaria przeciążenie prądowe
   RUNG wire#powerrail
      Contact( "AlwaysTRUE" )
      Contact( "IsCurrentOverloadInverter" )
      Move(in := "dbtags_Sterowanie".SetupControlPompownia.CurrentMax_Manual_Hz, out1 => "dbdane".Manual_SV)
   END_RUNG
   // the same network as SCL:
   IF "AlwaysTRUE" AND "IsCurrentOverloadInverter" THEN
       "dbdane".Manual_SV := "dbtags_Sterowanie".SetupControlPompownia.CurrentMax_Manual_Hz;
   END_IF;
END_REGION

REGION Network 17: Ustawienie tymczasowych Hz
   // Ustawienie tymczasowej wartości Hz
   RUNG wire#powerrail
      Contact( "Tmp_Set_SV" )
      Move(in := "dbTable of value Hz".Static_1[7], out1 => "dbdane".Manual_SV)
   END_RUNG
   // the same network as SCL:
   IF "Tmp_Set_SV" THEN "dbdane".Manual_SV := "dbTable of value Hz".Static_1[7]; END_IF;
END_REGION

REGION Network 18: Ustawienie bitu sygnały tymczasowej wartości Hz
   // Gdy Hz zadawane z PID są mniejsze od 15.0 Hz a zawartość bar mniejsza od zadanej i mniejsza od zera lub równa to ustaw wartość Hz tymczasową
   RUNG wire#powerrail
      I_Contact( "FirstScan" )
      I_Contact( "BarPress_Max" )
      I_Contact( "IsCurrentOverloadInverter" )
      Contact( "IEC_Timer_Reset_delay_DB".Q )
      { S7_Templates := "SrcType := Real" } LT_Contact(in1 := "dbdane".PV, in2 := "db10organizacyjna".setpoint_SV_bar)
      { S7_Templates := "SrcType := Real" } LE_Contact(in1 := "dbdane".OUT_PURE_Real, in2 := 15.0)
      S_Coil( "Tmp_Set_SV" )
   END_RUNG
   // the same network as SCL:
   IF NOT "FirstScan" AND NOT "BarPress_Max" AND NOT "IsCurrentOverloadInverter" AND "IEC_Timer_Reset_delay_DB".Q AND ("dbdane".PV < "db10organizacyjna".setpoint_SV_bar) AND ("dbdane".OUT_PURE_Real <= 15.0) THEN
       "Tmp_Set_SV" := TRUE;
   END_IF;
END_REGION

REGION Network 19: Reset znacznika ustawiania tymczasowej wartości Hz P1-P4
   RUNG wire#powerrail
      { S7_Templates := "SrcType := Real" } GE_Contact(in1 := "dbdane".OUT_PURE_Real, in2 := 16.0)
      wire#w1
      R_Coil( "Tmp_Set_SV" )
   END_RUNG
   RUNG wire#powerrail
      { S7_Templates := "SrcType := Real" } LE_Contact(in1 := "dbdane".PV, in2 := 0.0)
   END_RUNG wire#w1
   RUNG wire#powerrail
      Contact( "AlwaysTRUE" )
      { S7_Templates := "SrcType := Real" } GT_Contact(in1 := "dbdane".PV, in2 := "dbdane".Setpoint_SV)
   END_RUNG wire#w1
   // the same network as SCL:
   IF ("dbdane".OUT_PURE_Real >= 16.0) OR ("dbdane".PV <= 0.0) OR ("AlwaysTRUE" AND ("dbdane".PV > "dbdane".Setpoint_SV)) THEN
       "Tmp_Set_SV" := FALSE;
   END_IF;
END_REGION

REGION Network 20: Skalowanie wartości tymczasowych Hz to %QW P1-P4
   // "dane".Temp_SV - Tymczasowa wartość Hz  (30Hz)
   RUNG wire#powerrail
      Contact( "AlwaysTRUE" )
      Move(in := 8294, out1 => "dbdane".Temp_SV)
   END_RUNG
   // the same network as SCL:
   IF "AlwaysTRUE" THEN "dbdane".Temp_SV := 8294; END_IF;
END_REGION

REGION Network 21: Histerezas Reset Hz ustawionych manualnie
   RUNG wire#powerrail
      { S7_Templates := "SrcType := Real" } GE_Contact(in1 := "dbdane".OUT_PURE_Real, in2 := 10.0)
      { S7_Templates := "time_type := Time" } "IEC_Timer_Set_50Hz_DB".TON(pt := T#20S, et =>)
   END_RUNG
   // the same network as SCL:
   "IEC_Timer_Set_50Hz_DB".TON(IN := "dbdane".OUT_PURE_Real >= 10.0, PT := T#20S);
END_REGION

REGION Network 22: Reset znacznika płynnego przełaczenie Hz z tymczasowych na podawane z PID
   // Reset znacznika manualnego zadawania Hz
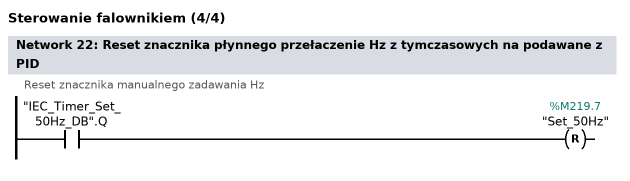
   RUNG wire#powerrail
      Contact( "IEC_Timer_Set_50Hz_DB".Q )
      R_Coil( "Set_50Hz" )
   END_RUNG
   // the same network as SCL:
   IF "IEC_Timer_Set_50Hz_DB".Q THEN "Set_50Hz" := FALSE; END_IF;
END_REGION
END_FUNCTION_BLOCK

FUNCTION_BLOCK "Sterowanie dołączeniem na sieć"   // FB10, LAD
TITLE = Sterowanie stycznikiem sieć
{ S7_Optimized_Access := 'TRUE' }
AUTHOR : rtecmer
VERSION : 0.1
// Sterowanie stycznikiem sieć. Ustawianie znaczników setCMD_SM i setSUPV_SM które przekazywane są do funkcji FC3/FC1 DRV01 driver napędów. Następnie przekazywane jest do warstwy Hardware/ OUT gdzie ustawiane jest wyjście sterownika
// stored: AutoNumber true, IsIECCheckEnabled false, IsRetainMemResEnabled false, MemoryReserve 500, SetENOAutomatically false, UDAEnableTagReadback false
   VAR_INPUT
      IsReady_M : Bool;   // Gotowość napędu
      IsModeAut : Bool;   // Znacznik tryb pracy
      Time_Off_Inverter : Bool;   // Bit Q - timer blokowania stycznika falownika po wyłączeniu / Bit Q - timer blokowania stycznika falownika po wyłaczeniu
      setMotor2 : Bool;   // Znacznik dodatkowa pompy nr1 / Znacznik dodatkowa dmuchawa nr1
      setMotor3 : Bool;   // Znacznik ustawienie dodatkowej 2 / Znacznik ustawienie dodatkowej dmuchawy nr 2
      setMotor4 : Bool;   // Znacznik ustawienie dodatkowej 3 / Znacznik ustawienie dodatkowej dmuchawy nr3
      IsRunNetwork_M : Bool;   // Potwierdzenie pracy z sieci M
      CMD_A_NetworkM : Bool;   // Znacznik serowania awaryjnego napędem z sieci w wypadku awarii falownika / Znacznikserowania awaryjnego napędem z sieci w wypadku awarii falownika
   END_VAR
   VAR_IN_OUT
      TimerStartNetworkContactor : TON_TIME;   // Opóżnienie załaczenia stycznika sieć
      setCMD_SM : Bool;   // Znacznik sterowania stycznikiem sieć / Znacznik sterowania w trybie sieć
      Is_extras_K1_M_1 : Bool;   // Znacznik motor dodatkowy nr 1
      Is_extras_K2_M_1 : Bool;   // Znacznik motor dodatkowy nr 2
      Is_extras_K3_M_1 : Bool;   // Znacznik motor dodatkowy nr 3
      setSUPV_SM : Bool;   // Znacznik polecenia sterowania z sieci / Znacznik polecenia startu z sieci
      off_add_K1 : Bool;   // znacznik pomocniczy podczas selektrywnego wyłączeania dodatkowej pompy
      off_add_K2 : Bool := false;   // znacznik pomocniczy podczas selektrywnego wyłączeania dodatkowej pompy
      off_add_K3 : Bool := false;   // znacznik pomocniczy podczas selektrywnego wyłączeania dodatkowej pompy
   END_VAR
   VAR_TEMP
      tmpOFFinverter : Bool;   // wyłączenie od osiągnięcia 50Hz + czas zwłoki
      mem_activ_K1 : Bool;   // pamięć załączennie jako dodatkowa
      mem_activ_K2 : Bool;   // pamięć załączennie jako dodatkowa
      mem_activ_K3 : Bool;   // pamięć załączennie jako dodatkowa
   END_VAR
   VAR_TEMP   // added for the SCL form of the ladder/FBD networks
      _w1 : Bool;
   END_VAR
BEGIN

REGION Network 1: Timer opóźnienie dołączenie stycznika sieci
   // Histereza na dołączenie stycznika sieć po pracy z falownika
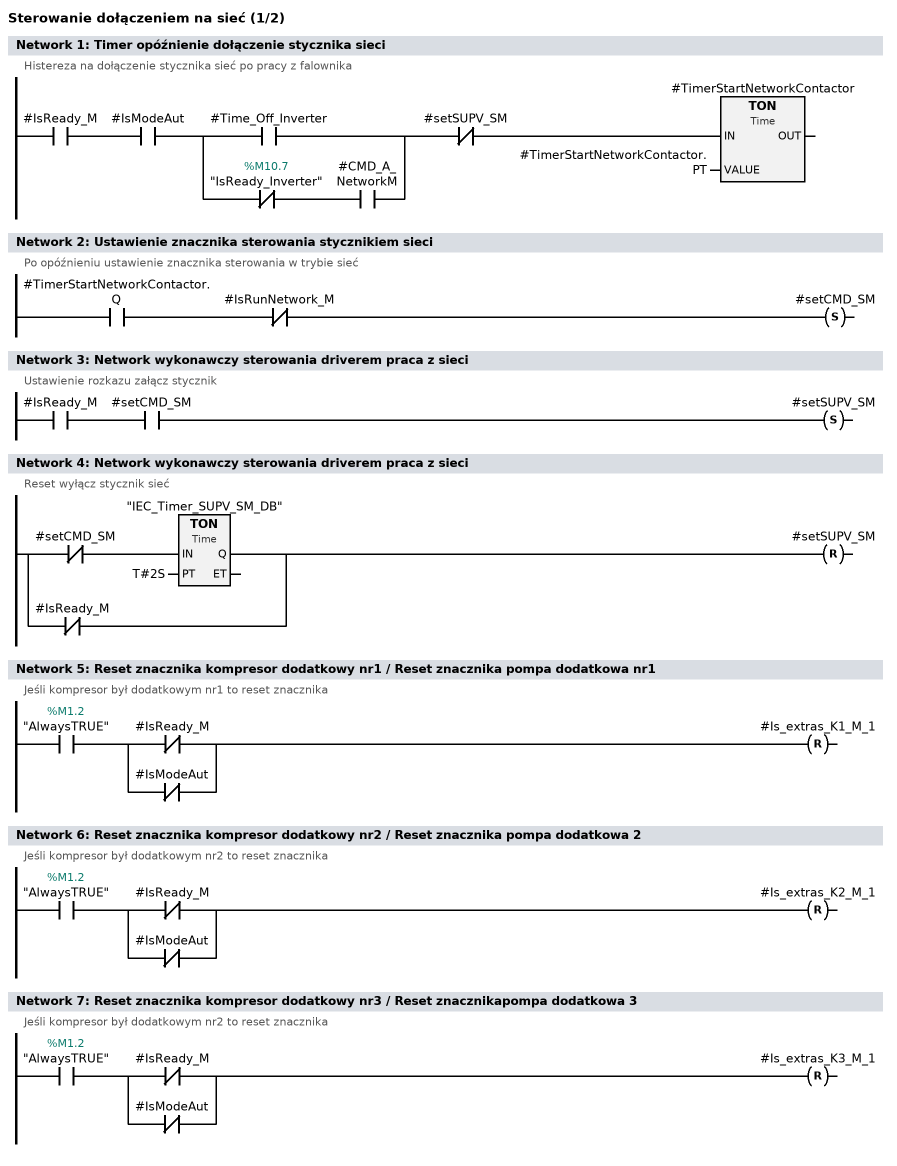
   #TimerStartNetworkContactor(IN := #IsReady_M AND #IsModeAut AND (#Time_Off_Inverter OR (NOT "IsReady_Inverter" AND #CMD_A_NetworkM)) AND NOT #setSUPV_SM, PT := #TimerStartNetworkContactor.PT);   // TON coil
END_REGION

REGION Network 2: Ustawienie znacznika sterowania stycznikiem sieci
   // Po opóźnieniu ustawienie znacznika sterowania w trybie sieć
   RUNG wire#powerrail
      Contact( #TimerStartNetworkContactor.Q )
      I_Contact( #IsRunNetwork_M )
      S_Coil( #setCMD_SM )
   END_RUNG
   // the same network as SCL:
   IF #TimerStartNetworkContactor.Q AND NOT #IsRunNetwork_M THEN #setCMD_SM := TRUE; END_IF;
END_REGION

REGION Network 3: Network wykonawczy sterowania driverem praca z sieci
   // Ustawienie rozkazu załącz stycznik
   RUNG wire#powerrail
      Contact( #IsReady_M )
      Contact( #setCMD_SM )
      S_Coil( #setSUPV_SM )
   END_RUNG
   // the same network as SCL:
   IF #IsReady_M AND #setCMD_SM THEN #setSUPV_SM := TRUE; END_IF;
END_REGION

REGION Network 4: Network wykonawczy sterowania driverem praca z sieci
   // Reset wyłącz stycznik sieć
   RUNG wire#powerrail
      I_Contact( #setCMD_SM )
      { S7_Templates := "time_type := Time" } "IEC_Timer_SUPV_SM_DB".TON(pt := T#2S, et =>)
      wire#w1
      R_Coil( #setSUPV_SM )
   END_RUNG
   RUNG wire#powerrail
      I_Contact( #IsReady_M )
   END_RUNG wire#w1
   // the same network as SCL:
   "IEC_Timer_SUPV_SM_DB".TON(IN := NOT #setCMD_SM, PT := T#2S);
   IF "IEC_Timer_SUPV_SM_DB".Q OR NOT #IsReady_M THEN #setSUPV_SM := FALSE; END_IF;
END_REGION

REGION Network 5: Reset znacznika kompresor dodatkowy nr1 / Reset znacznika pompa dodatkowa nr1
   // Jeśli kompresor był dodatkowym nr1 to reset znacznika
   RUNG wire#powerrail
      Contact( "AlwaysTRUE" )
      wire#w1
      I_Contact( #IsReady_M )
      wire#w2
      R_Coil( #Is_extras_K1_M_1 )
   END_RUNG
   RUNG wire#w1
      I_Contact( #IsModeAut )
   END_RUNG wire#w2
   // the same network as SCL:
   IF "AlwaysTRUE" AND (NOT #IsReady_M OR NOT #IsModeAut) THEN #Is_extras_K1_M_1 := FALSE; END_IF;
END_REGION

REGION Network 6: Reset znacznika kompresor dodatkowy nr2 / Reset znacznika pompa dodatkowa 2
   // Jeśli kompresor był dodatkowym nr2 to reset znacznika
   RUNG wire#powerrail
      Contact( "AlwaysTRUE" )
      wire#w1
      I_Contact( #IsReady_M )
      wire#w2
      R_Coil( #Is_extras_K2_M_1 )
   END_RUNG
   RUNG wire#w1
      I_Contact( #IsModeAut )
   END_RUNG wire#w2
   // the same network as SCL:
   IF "AlwaysTRUE" AND (NOT #IsReady_M OR NOT #IsModeAut) THEN #Is_extras_K2_M_1 := FALSE; END_IF;
END_REGION

REGION Network 7: Reset znacznika kompresor dodatkowy nr3 / Reset znacznikapompa dodatkowa 3
   // Jeśli kompresor był dodatkowym nr2 to reset znacznika
   RUNG wire#powerrail
      Contact( "AlwaysTRUE" )
      wire#w1
      I_Contact( #IsReady_M )
      wire#w2
      R_Coil( #Is_extras_K3_M_1 )
   END_RUNG
   RUNG wire#w1
      I_Contact( #IsModeAut )
   END_RUNG wire#w2
   // the same network as SCL:
   IF "AlwaysTRUE" AND (NOT #IsReady_M OR NOT #IsModeAut) THEN #Is_extras_K3_M_1 := FALSE; END_IF;
END_REGION

REGION Network 8: Reset Znacznika sterowania w trybie sieć
   // Gdy regulator PID ustawi szybkie wyłaczenie pompy dodatkowej nr , n2 to następuje resetowania znacznika pracy pompy dodatkowej / Gdy regulator PID ustawi szybkie wyłaczenie pompy dodatkowej nr 1, nr 2, nr 3 to następuje resetowania znacznika pracy pompy dodatkowej
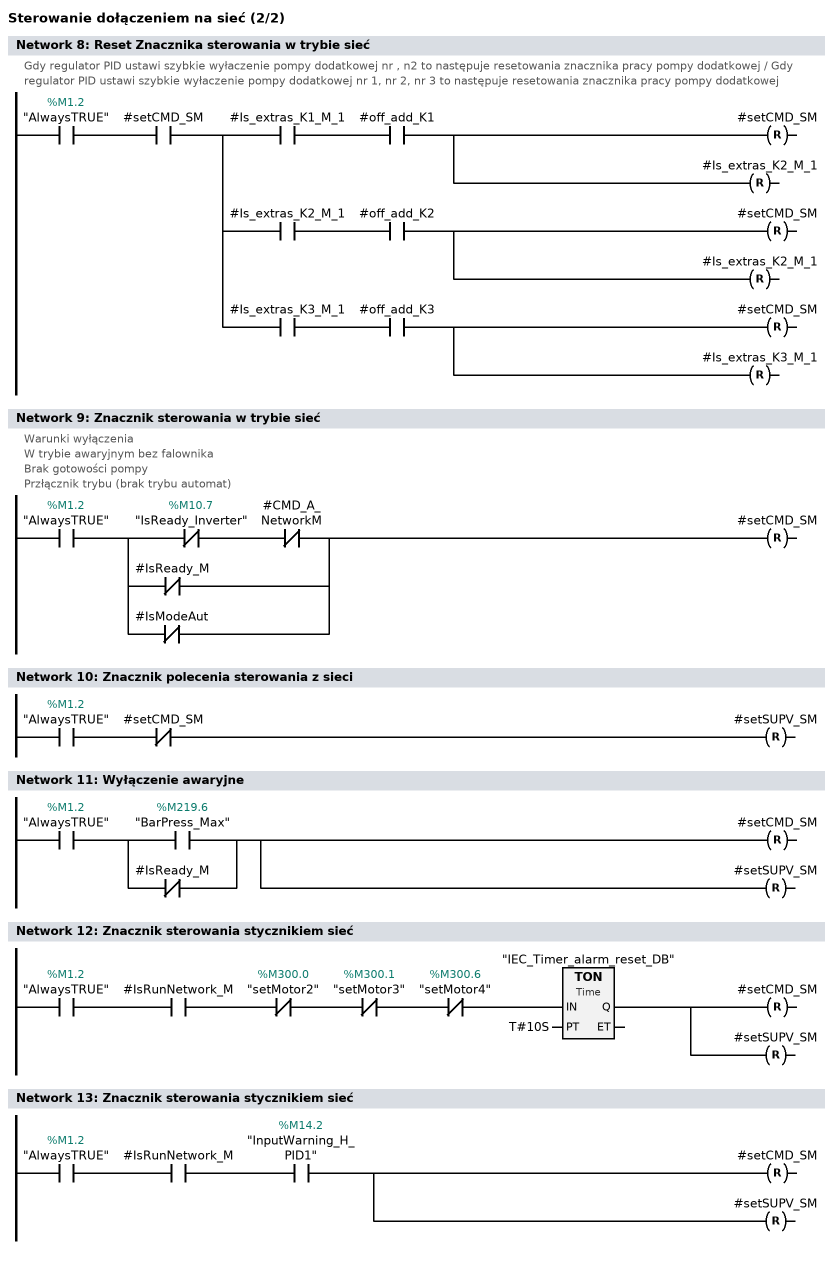
   RUNG wire#powerrail
      Contact( "AlwaysTRUE" )
      Contact( #setCMD_SM )
      wire#w1
      Contact( #Is_extras_K1_M_1 )
      Contact( #off_add_K1 )
      wire#w2
      R_Coil( #setCMD_SM )
   END_RUNG
   RUNG wire#w2
      R_Coil( #Is_extras_K2_M_1 )
   END_RUNG
   RUNG wire#w1
      Contact( #Is_extras_K2_M_1 )
      Contact( #off_add_K2 )
      wire#w3
      R_Coil( #setCMD_SM )
   END_RUNG
   RUNG wire#w3
      R_Coil( #Is_extras_K2_M_1 )
   END_RUNG
   RUNG wire#w1
      Contact( #Is_extras_K3_M_1 )
      Contact( #off_add_K3 )
      wire#w4
      R_Coil( #setCMD_SM )
   END_RUNG
   RUNG wire#w4
      R_Coil( #Is_extras_K3_M_1 )
   END_RUNG
   // the same network as SCL:
   #_w1 := "AlwaysTRUE" AND #setCMD_SM;
   IF #_w1 AND #Is_extras_K1_M_1 AND #off_add_K1 THEN
       #setCMD_SM := FALSE;
       #Is_extras_K2_M_1 := FALSE;
   END_IF;
   IF #_w1 AND #Is_extras_K2_M_1 AND #off_add_K2 THEN
       #setCMD_SM := FALSE;
       #Is_extras_K2_M_1 := FALSE;
   END_IF;
   IF #_w1 AND #Is_extras_K3_M_1 AND #off_add_K3 THEN
       #setCMD_SM := FALSE;
       #Is_extras_K3_M_1 := FALSE;
   END_IF;
END_REGION

REGION Network 9: Znacznik sterowania w trybie sieć
   // Warunki wyłączenia 
   // W trybie awaryjnym bez falownika
   // Brak gotowości pompy
   // Przłącznik trybu (brak trybu automat)
   RUNG wire#powerrail
      Contact( "AlwaysTRUE" )
      wire#w1
      I_Contact( "IsReady_Inverter" )
      I_Contact( #CMD_A_NetworkM )
      wire#w2
      R_Coil( #setCMD_SM )
   END_RUNG
   RUNG wire#w1
      I_Contact( #IsReady_M )
   END_RUNG wire#w2
   RUNG wire#w1
      I_Contact( #IsModeAut )
   END_RUNG wire#w2
   // the same network as SCL:
   IF "AlwaysTRUE" AND ((NOT "IsReady_Inverter" AND NOT #CMD_A_NetworkM) OR NOT #IsReady_M OR NOT #IsModeAut) THEN
       #setCMD_SM := FALSE;
   END_IF;
END_REGION

REGION Network 10: Znacznik polecenia sterowania z sieci
   RUNG wire#powerrail
      Contact( "AlwaysTRUE" )
      I_Contact( #setCMD_SM )
      R_Coil( #setSUPV_SM )
   END_RUNG
   // the same network as SCL:
   IF "AlwaysTRUE" AND NOT #setCMD_SM THEN #setSUPV_SM := FALSE; END_IF;
END_REGION

REGION Network 11: Wyłączenie awaryjne
   RUNG wire#powerrail
      Contact( "AlwaysTRUE" )
      wire#w1
      Contact( "BarPress_Max" )
      wire#w2
      R_Coil( #setCMD_SM )
   END_RUNG
   RUNG wire#w1
      I_Contact( #IsReady_M )
   END_RUNG wire#w2
   RUNG wire#w2
      R_Coil( #setSUPV_SM )
   END_RUNG
   // the same network as SCL:
   IF "AlwaysTRUE" AND ("BarPress_Max" OR NOT #IsReady_M) THEN
       #setCMD_SM := FALSE;
       #setSUPV_SM := FALSE;
   END_IF;
END_REGION

REGION Network 12: Znacznik sterowania stycznikiem sieć
   RUNG wire#powerrail
      Contact( "AlwaysTRUE" )
      Contact( #IsRunNetwork_M )
      I_Contact( "setMotor2" )
      I_Contact( "setMotor3" )
      I_Contact( "setMotor4" )
      { S7_Templates := "time_type := Time" } "IEC_Timer_alarm_reset_DB".TON(pt := T#10S, et =>)
      wire#w1
      R_Coil( #setCMD_SM )
   END_RUNG
   RUNG wire#w1
      R_Coil( #setSUPV_SM )
   END_RUNG
   // the same network as SCL:
   "IEC_Timer_alarm_reset_DB".TON(IN := "AlwaysTRUE" AND #IsRunNetwork_M AND NOT "setMotor2" AND NOT "setMotor3" AND NOT "setMotor4",
                           PT := T#10S);
   IF "IEC_Timer_alarm_reset_DB".Q THEN
       #setCMD_SM := FALSE;
       #setSUPV_SM := FALSE;
   END_IF;
END_REGION

REGION Network 13: Znacznik sterowania stycznikiem sieć
   RUNG wire#powerrail
      Contact( "AlwaysTRUE" )
      Contact( #IsRunNetwork_M )
      Contact( "InputWarning_H_PID1" )
      wire#w1
      R_Coil( #setCMD_SM )
   END_RUNG
   RUNG wire#w1
      R_Coil( #setSUPV_SM )
   END_RUNG
   // the same network as SCL:
   IF "AlwaysTRUE" AND #IsRunNetwork_M AND "InputWarning_H_PID1" THEN
       #setCMD_SM := FALSE;
       #setSUPV_SM := FALSE;
   END_IF;
END_REGION
END_FUNCTION_BLOCK

FUNCTION "Komutacja Styczników_Sygnałów" : Void
TITLE = Blok sterowania stycznikami F/S i sygnał ON/OFF Soft-Start/ Falo
{ S7_Optimized_Access := 'TRUE' }
AUTHOR : rtecmer
VERSION : 0.1
//Funkcja służy do sterowania stycznikami sieć, falownik napędów P1-P4. 

BEGIN
	(*
	//=============================================================================
	//(JZWiK S.A Radosław Tecmer)
	//(c)Copyright (2021) All Rights Reserved
	//-----------------------------------------------------------------------------
	//Testowane z:   (system docelowy z  FW 4.4)
	//Pakiet inżynierski:   TIA Portal (V14 Sp1 Update 9)
	//Ograniczenia:  ( - )
	//Wymagania:  (minimalne S7-1200 CPU 1215C FW 4.2 .)
	//Funkcjonalnośc: (Komutacja styczników F/S. Sterowanie sygnałami On/Off soft-start
	//                i falownik)
	//-----------------------------------------------------------------------------
	//Zmainy wprowadzone:
	//Wersja  Data       Osoba wprowadzająca zmiany - ekspert
	//01.00.00 09.1.2022 (Tecmer Radosław - twórca) Pieresza wersja 01.00.00
	//=============================================================================
	*)
	
	
	
	REGION Pompa P1 
	  // sterowanie stycznikami falownik
	  IF ("CB_CMD_P1" = 1) AND ("IsReady_P1" = 1) AND
	    ("setCMD_FP1" = 1) AND
	    ("CMD_network_P1" = 0) AND
	    ("CMD_inverter_P2" = 0) AND ("CMD_inverter_P3" = 0) AND ("CMD_inverter_P4" = 0)
	  THEN
	    // Sterowanie stycznikiem falownika 
	    "CMD_inverter_P1" := TRUE;
	  ELSE
	    "CMD_inverter_P1" := FALSE;
	    ;
	  END_IF;
	  
	
	  
	  // Sterowanie stycznikiem sieć 
	  IF (("CB_CMD_P1" = 1) AND ("IsReady_P1" = 1) AND
	    ("setCMD_SP1" = 1) AND
	    ("CMD_inverter_P1" = 0))
	    OR
	    ("CB_CMD_P1" = 1 AND "bitH_Aut_Man_P1" = 0 AND "CMD_inverter_P1" = 0)
	  THEN
	    // Sterowanie stycznikiem sieć 
	    "CMD_network_P1" := TRUE;
	  ELSE
	    "CMD_network_P1" := FALSE;
	    ;
	  END_IF;
	  
	 
	  
	  // Sterowanie sygnałem podawanym na Soft-Start
	  IF "inputRunS_P1" AND "bitH_Alarm_P1"= FALSE AND  "IsRem" THEN
	    // Podaj sybnał start na soft-start
	    "CMD_soft_P1" := "CMD_network_P1";
	  ELSE
	    "CMD_soft_P1" := FALSE;
	    ;
	  END_IF;
	  
	  
	  
	END_REGION
	
	REGION Pompa P2
	  // sterowanie stycznikami falownik
	  IF ("CB_CMD_P2" = 1) AND ("IsReady_P2" = 1) AND
	    ("setCMD_FP2" = 1) AND
	    ("CMD_network_P2" = 0) AND
	    ("CMD_inverter_P1" = 0) AND ("CMD_inverter_P3" = 0) AND ("CMD_inverter_P4" = 0)
	  THEN
	    // Sterowanie stycznikiem falownika
	    "CMD_inverter_P2" := TRUE;
	  ELSE
	    "CMD_inverter_P2" := FALSE;
	    ;
	  END_IF;
	  
	
	  
	  // Sterowanie stycznikiem sieć 
	  IF (("CB_CMD_P2" = 1) AND ("IsReady_P2" = 1) AND
	    ("setCMD_SP2" = 1) AND
	    ("CMD_inverter_P2" = 0))
	    OR
	    ("CB_CMD_P2" = 1 AND "bitH_Aut_Man_P2" = 0 AND "CMD_inverter_P2" = 0 )
	  THEN
	    // Sterowanie stycznikiem sieć 
	    "CMD_network_P2" := TRUE;
	  ELSE
	    "CMD_network_P2" := FALSE;
	    ;
	  END_IF;
	  
	 
	  
	  // Sterowanie sygnałem podawanym na Soft-Start
	  IF "inputRunS_P2" AND "bitH_Alarm_P2"= FALSE AND  "IsRem" THEN
	    // Podaj sybnał start na soft-start
	    "CMD_soft_P2" := "CMD_network_P2";
	  ELSE
	    "CMD_soft_P2" := FALSE;
	    ;
	  END_IF;
	  
	  
	END_REGION
	
	REGION Pompa P3
	  // sterowanie stycznikami falownik
	  IF ("CB_CMD_P3" = 1) AND ("IsReady_P3" = 1) AND
	    ("setCMD_FP3" = 1) AND
	    ("CMD_network_P3" = 0) AND
	    ("CMD_inverter_P2" = 0) AND ("CMD_inverter_P1" = 0) AND ("CMD_inverter_P4" = 0)
	  THEN
	    // Sterowanie stycznikiem falownika 
	    "CMD_inverter_P3" := TRUE;
	  ELSE
	    "CMD_inverter_P3" := FALSE;
	    ;
	  END_IF;
	  
	 
	  
	  // Sterowanie stycznikiem sieć 
	  IF (("CB_CMD_P3" = 1) AND ("IsReady_P3" = 1) AND
	    ("setCMD_SP3" = 1) AND
	    ("CMD_inverter_P3" = 0))
	    OR
	    ("CB_CMD_P3" = 1 AND "bitH_Aut_Man_P3" = 0 AND "CMD_inverter_P3" = 0)
	  THEN
	     //Sterowanie stycznikiem sieć 
	    "CMD_network_P3" := TRUE;
	  ELSE
	    "CMD_network_P3" := FALSE;
	    ;
	  END_IF;
	  
	 
	  
	  // Sterowanie sygnałem podawanym na Soft-Start
	  IF "inputRunS_P3" AND "bitH_Alarm_P3"= FALSE AND  "IsRem" THEN
	     //Podaj sybnał start na soft-start
	    "CMD_soft_P3" := "CMD_network_P3";
	  ELSE
	    "CMD_soft_P3":= FALSE;
	    ;
	  END_IF;
	  
	  
	END_REGION
	
	
	
	REGION Pompa P4
	  // sterowanie stycznikami falownik
	  IF ("CB_CMD_P4" = 1) AND ("IsReady_P4" = 1) AND
	    ("setCMD_FP4" = 1) AND
	    ("CMD_network_P4" = 0) AND
	    ("CMD_inverter_P2" = 0) AND ("CMD_inverter_P1" = 0) AND ("CMD_inverter_P3" = 0)
	  THEN
	    // Sterowanie stycznikiem falownika 
	    "CMD_inverter_P4" := TRUE;
	  ELSE
	    "CMD_inverter_P4" := FALSE;
	    ;
	  END_IF;
	  
	  
	  IF (("CB_CMD_P4" = 1) AND ("IsReady_P4" = 1) AND
	    ("setCMD_SP4" = 1) AND
	    ("CMD_inverter_P4" = 0))
	    OR
	    ("CB_CMD_P4" = 1 AND "bitH_Aut_Man_P4" = 0 AND "CMD_inverter_P4" = 0)
	  THEN
	    // Sterowanie stycznikiem sieć 
	    "CMD_network_P4" := TRUE;
	  ELSE
	    "CMD_network_P4" := FALSE;
	    ;
	  END_IF;
	  
	
	  
	  
	  // Sterowanie sygnałem podawanym na Soft-Start
	  IF "inputRunS_P4" AND "bitH_Alarm_P4"= FALSE AND  "IsRem" THEN
	    // Podaj sybnał start na soft-start
	    "CMD_soft_P4" := "CMD_network_P4";
	  ELSE
	    "CMD_soft_P4" := FALSE;
	    ;
	  END_IF;
	  
	END_REGION
END_FUNCTION

FUNCTION "OUT" : Void
TITLE = OUT 
{ S7_Optimized_Access := 'TRUE' }
AUTHOR : rtecmer
VERSION : 0.1
//Mapowamie i wyzwalanie wyjść 

BEGIN
	(*
	Sterowanie przekaźnikami sieć, falownik pompy 
	Sprawdzanie wyjść sterowniak i przekazanie sygnałów 
	*)
	
	
	
	REGION Sygnalizacja Awarii
	  
	  // Wijścia przekaźnikowe sygnalizacja awarii
	  //Pomp Zasuw Falownika Soft-start
	  "Q3.5" := "CMD_faultInverter";
	  "Q0.3" := "CMD_faultP1";
	  "Q0.7" := "CMD_faultP2";
	  "Q2.1" := "CMD_faultP3";
	  "Q2.5" := "CMD_faultP4";
	  
	END_REGION
	
	REGION "inverter"
	  // Przekazanie wartości
	  "Q2.6" := "CMD_start_stop_inverter";
	  
	END_REGION
	
	
	REGION Styczniki P1
	  // Przekazanie wartości
	  "Q0.1" := "CMD_inverter_P1";
	  "Q0.0" := "CMD_network_P1";
	  "Q0.2" := "CMD_soft_P1";
	  "Q4.0" := "resetFault_SoftStart_P1";
	 
	END_REGION
	
	REGION Styczniki P2
	  // Przekazanie wartości
	  "Q0.5" := "CMD_inverter_P2";
	  "Q0.4" := "CMD_network_P2";
	  "Q0.6" := "CMD_soft_P2";
	  "Q4.1" := "resetFault_SoftStart_P2";
	  
	END_REGION
	
	REGION Styczniki P3
	  // Przekazanie wartości
	  "Q1.1" := "CMD_inverter_P3";
	  "Q1.0" := "CMD_network_P3";
	  "Q2.0" := "CMD_soft_P3";
	  "Q4.2" := "resetFault_SoftStart_P3";
	  
	END_REGION
	
	REGION Styczniki P4
	  // Przekazanie wartości
	  "Q2.3" := "CMD_inverter_P4";
	  "Q2.2" := "CMD_network_P4";
	  "Q2.4" := "CMD_soft_P4";
	  "Q4.3" := "resetFault_SoftStart_P4";
	  
	END_REGION
	
	REGION Zasuwa Z11
	  // Przekazanie wartości
	  //Otwieranie
	  "Q2.7" := "CMD_Open_Z11";
	  //Zamykanie
	  "Q3.0" := "CMD_Close_Z11";
	  // Awaria
	  "Q3.1" := NOT("isReadyZ11");
	  
	END_REGION
	
	REGION Zasuwa Z12
	  // Przekazanie wartości
	  //Otwieranie
	  "Q3.2" := "CMD_Open_Z12";
	  //Zamykanie
	  "Q3.3" := "CMD_Close_Z12";
	  //Awaria
	 
	  "Q3.4" := NOT("isReadyZ12");
	  
	END_REGION
	  
	
	
	
	
	
	
	
	
	
	
	 
	
	
	
	
	 
	 
	
	 
	 
	 
END_FUNCTION

FUNCTION "Write_to DB_HoldReg_MT101" : Void
{ S7_Optimized_Access := 'TRUE' }
AUTHOR : rtecmer
VERSION : 0.1

BEGIN
	(*
	//=============================================================================
	//(JZWiK S.A Radosław Tecmer)
	//(c)Copyright (2021) All Rights Reserved
	//-----------------------------------------------------------------------------
	//Testowane z:   (system docelowy z  FW 4.2)
	//Pakiet inżynierski:   TIA Portal (V14 Sp1 Update 9)
	//Ograniczenia:  ( - )
	//Wymagania:  (minimalne S7-1200 CPU 1214 FW 3.2 .)
	//Funkcjonalnośc: (Kopiowanie bloków danych )
	//-----------------------------------------------------------------------------
	//Zmainy wprowadzone:
	//Wersja  Data       Osoba wprowadzająca zmiany - ekspert
	//01.00.00 17.11.2021 (Tecmer Radosław - twórca) Pieresza wersja 01.00.00
	//=============================================================================
	*)
	
	
	
	REGION  Stacja Zasów Status Napędów
	  // PLC Zasówy z modbus TCP
	  "db10organizacyjna".instvValveZ1 := "dbHold_RRG".status_Z1;
	  "db10organizacyjna".instvValveZ2 := "dbHold_RRG".status_Z2;
	  "db10organizacyjna".instvValveZ3 := "dbHold_RRG".status_Z3;
	  "db10organizacyjna".instvValveZ4 := "dbHold_RRG".status_Z4;
	  "db10organizacyjna".instvValveZ5 := "dbHold_RRG".status_Z5;
	  "db10organizacyjna".instvValveZ6 := "dbHold_RRG".status_Z6;
	  "db10organizacyjna".instvValveZ7 := "dbHold_RRG".status_Z7;
	  "db10organizacyjna".instvValveZ8 := "dbHold_RRG".status_Z8;
	  "db10organizacyjna".instvValveZ9 := "dbHold_RRG".status_Z9;
	  "db10organizacyjna".instvValveZ10 := "dbHold_RRG".status_Z10;
	  
	  // Do instancji SCADA na MT101
	  "dbHoldRegSlave_to_MT101".instvValveZ1 := "db10organizacyjna".instvValveZ1;
	  "dbHoldRegSlave_to_MT101".instvValveZ2 := "db10organizacyjna".instvValveZ2;
	  "dbHoldRegSlave_to_MT101".instvValveZ3 := "db10organizacyjna".instvValveZ3;
	  "dbHoldRegSlave_to_MT101".instvValveZ4 := "db10organizacyjna".instvValveZ4;
	  "dbHoldRegSlave_to_MT101".instvValveZ5 := "db10organizacyjna".instvValveZ5;
	  "dbHoldRegSlave_to_MT101".instvValveZ6 := "db10organizacyjna".instvValveZ6;
	  "dbHoldRegSlave_to_MT101".instvValveZ7 := "db10organizacyjna".instvValveZ7;
	  "dbHoldRegSlave_to_MT101".instvValveZ8 := "db10organizacyjna".instvValveZ8;
	  "dbHoldRegSlave_to_MT101".instvValveZ9 := "db10organizacyjna".instvValveZ9;
	  "dbHoldRegSlave_to_MT101".instvValveZ10 := "db10organizacyjna".instvValveZ10;
	  
	END_REGION
	
	REGION Z10 położenie
	  //aktualne
	  "db10organizacyjna".actPozycja_Z10 := "dbHold_RRG".act_położenie_Z10;
	  "dbHoldRegSlave_to_MT101".instPozitionZ10_act:= INT_TO_REAL ("db10organizacyjna".actPozycja_Z10);
	END_REGION
	
	REGION Analogi
	  // Przekazanie
	  "dbHoldRegSlave_to_MT101".instB5bar_act := "db10organizacyjna".instB5_bar_act_magistrala;
	  "dbHoldRegSlave_to_MT101".instB6bar_act := "db10organizacyjna".instB6_bar_act_miasto;
	  "dbHoldRegSlave_to_MT101".instB7bar_act := "db10organizacyjna".instB7_bar_act_pompownia;
	  "dbHoldRegSlave_to_MT101".instB8bar_act := "dbdane".act_Value_B8;
	  "dbHoldRegSlave_to_MT101".instFlowDN225_act := "db10organizacyjna".instFlowDN225_act_Q1;
	  "dbHoldRegSlave_to_MT101".instFlowDN225_sum := "db10organizacyjna".instSumFlowDN225_Q1;
	  "dbHoldRegSlave_to_MT101".instFlowDN500_act := "db10organizacyjna".instFlowDN500_act_Q2;
	  "dbHoldRegSlave_to_MT101".instFlowDN500_sum := "db10organizacyjna".instSumFlowDN500_Q2;
	  "dbHoldRegSlave_to_MT101".instCurrent_Inverter := REAL_TO_INT("db10organizacyjna".inst_act_Current_Inverters);
	  "dbHoldRegSlave_to_MT101".instHz_Inverter := REAL_TO_INT("db10organizacyjna".act_Hz_Inverter_1);
	  "dbHold_RRG".Sending.set_magistrala_alarm_min_bar := "dbHoldRegSlave_to_MT101".instSetBarMinB9;
	  // Magistrala zasilająca DN 500
	  // aktualny
	  "dbHoldRegSlave_to_MT101".instFlowDN500_act := "dbHold_RRG".act_przepływ_VF_Q2;
	  //Suma
	  "dbHoldRegSlave_to_MT101".instFlowDN500_sum := "dbHold_RRG".sum_przepływ_Q2;
	  // Miasto DN225
	  // aktualny
	  
	  "dbHoldRegSlave_to_MT101".instFlowDN225_act := "dbModbusRTU_Reg"."Przepływomierz nr1 pompownia".received_5_przeływu_VF_Adres_0;
	  //Suma
	  "dbHoldRegSlave_to_MT101".instFlowDN225_sum := "dbModbusRTU_Reg"."Przepływomierz nr1 pompownia".received_5_objętość_VF_Adres_2;
	END_REGION
	
	REGION Poziom w zbiornikach
	  // przekazanie
	  "dbHoldRegSlave_to_MT101".instLevelTank1 := REAL_TO_INT ("dbHold_RRG".act_poziom_ZB1);
	  "dbHoldRegSlave_to_MT101".instLevelTank2 := REAL_TO_INT ("dbHold_RRG".act_poziom_ZB2);
	  "dbHoldRegSlave_to_MT101".instLevelTank3 := REAL_TO_INT ("dbHold_RRG".act_poziom_ZB3);
	  "dbHoldRegSlave_to_MT101".instLevelTank4 := REAL_TO_INT ("dbHold_RRG".act_poziom_ZB4);
	  
	  
	END_REGION
	
	
	
	
	
	
	
END_FUNCTION

FUNCTION "Conroll_from_ModbusRTU" : Void
{ S7_Optimized_Access := 'TRUE' }
AUTHOR : rtecmer
VERSION : 0.1

BEGIN
	(*
	//=============================================================================
	//(JZWiK S.A Radosław Tecmer)
	//(c)Copyright (2021) All Rights Reserved
	//-----------------------------------------------------------------------------
	//Testowane z:   (system docelowy z  FW 4.2)
	//Pakiet inżynierski:   TIA Portal (V14 Sp1 Update 9)
	//Ograniczenia:  ( - )
	//Wymagania:  (minimalne S7-1200 CPU 1214 FW 3.2 .)
	//Funkcjonalnośc: (Przesuniecie bajtów (podobnie do funkcji SWAP) 
	//                  i przekazanie do bloku danych pomiary z przepływomierza )
	//-----------------------------------------------------------------------------
	//Zmainy wprowadzone:
	//Wersja  Data       Osoba wprowadzająca zmiany - ekspert
	//01.00.00 17.11.2021 (Tecmer Radosław - twórca) Pieresza wersja 01.00.00
	//=============================================================================
	*)
	
	
	
	REGION Q1 przepływomierz
	  // Adres 0 - bierzący przepływ
	  "dbModbusRTU_Reg"."Przepływomierz nr1 pompownia".received_5_przeływu_VF_Adres_0 := DWORD_TO_REAL(%DB37.DBD0);
	 
	  "dbdane".Wielkość_przeływu_Q1 := "dbModbusRTU_Reg"."Przepływomierz nr1 pompownia".received_5_przeływu_VF_Adres_0;
	  
	  // Adres 2 - Licznik_objętość_VF
	  "dbModbusRTU_Reg"."Przepływomierz nr1 pompownia".received_5_objętość_VF_Adres_2 := DWORD_TO_REAL(%DB37.DBD4);
	  
	  "dbdane".Licznik_objętość_VF_Q1 := "dbModbusRTU_Reg"."Przepływomierz nr1 pompownia".received_5_objętość_VF_Adres_2;
	  
	  // Adres 4- stan bierzący licznika objetości w stecz VR
	  "dbModbusRTU_Reg"."Przepływomierz nr1 pompownia"."received_5_objętośc RF_Adres_4" := DWORD_TO_REAL(%DB37.DBD8);
	  
	  "dbdane".Licznik_objętość_VR_Q1 := "dbModbusRTU_Reg"."Przepływomierz nr1 pompownia"."received_5_objętośc RF_Adres_4";
	  
	  // Adres 6- stan bierzący licznika różnicowego  objętości VD
	  // 
	  "tmp_differential counter VD_H_Q1" := "dbModbusRTU_Reg".received_5_Licznik_różnicowy_VD_Adres_6.data[0];
	  "tmp_differential counter VD_L_Q1" := "dbModbusRTU_Reg".received_5_Licznik_różnicowy_VD_Adres_6.data[1];
	  "dbdane".Licznik_różnicowy_VD_Q1 := "act_differential counter VD_Q1";
	  
	  // Adres 8- główny liczni objetości w przód GF
	  "dbModbusRTU_Reg"."Przepływomierz nr1 pompownia".received_5_licznik_objętości_GF_Adres_8 := DWORD_TO_REAL(%DB37.DBD16);
	  
	  "dbdane".Stan_licz_bjętości_GF_Q1 := "dbModbusRTU_Reg"."Przepływomierz nr1 pompownia".received_5_licznik_objętości_GF_Adres_8;
	  
	  // Adres 10- główny liczni objetości w stecz GR
	  "dbModbusRTU_Reg"."Przepływomierz nr1 pompownia".received_5_Licznik_objętości_GR_Adres_10 := DWORD_TO_REAL(%DB37.DBD20);
	  
	  "dbdane".Stan_licz_rózicowego_obj_GD_Q1 := "dbModbusRTU_Reg"."Przepływomierz nr1 pompownia".received_5_Licznik_objętości_GR_Adres_10;
	  
	  //Adres 12- główny różnica liczni objetościGD
	  "tmp_differential counter status_GD_H_Q1" := "dbModbusRTU_Reg".received_5_Stan_licz_rózicowego_obj_GD_Adres_12.data[0];
	  "tmp_differential counter status_GD_L_Q1" := "dbModbusRTU_Reg".received_5_Stan_licz_rózicowego_obj_GD_Adres_12.data[1];
	  
	  // Status MP04 Q1 - pompownia
	  "dbModbusRTU_Reg"."Przepływomierz nr1 pompownia".received_5_status_przepływomierza_Adres_1000 := "dbModbusRTU_Reg".received_5_Stan_urządzenia_1000.typeDataInverter_int[0];
	  "dbdane"._Stan_urządzenia_Q1 := "dbModbusRTU_Reg".received_5_Stan_urządzenia_1000.typeDataInverter_int[0];
	END_REGION
	
	
	
	  
	  
	  
	  
	  
	  
	
	
END_FUNCTION

ORGANIZATION_BLOCK "Cyclic interrupt"   // OB30, LAD, CyclicInterrupt
{ S7_Optimized_Access := 'TRUE' }
AUTHOR : RTecmer
VERSION : 0.1
// stored: AutoNumber true, IsIECCheckEnabled false, SetENOAutomatically false
   VAR_TEMP
      Temp_SV_Int : Int;
      PV_Temp : Real;
      Temp_1 : Real;
   END_VAR
   VAR_TEMP   // added for the SCL form of the ladder/FBD networks
      _w1 : Bool;
      _w2 : Bool;
   END_VAR
BEGIN

REGION Network 1: WatchDog HMI
   // Do zrobienia
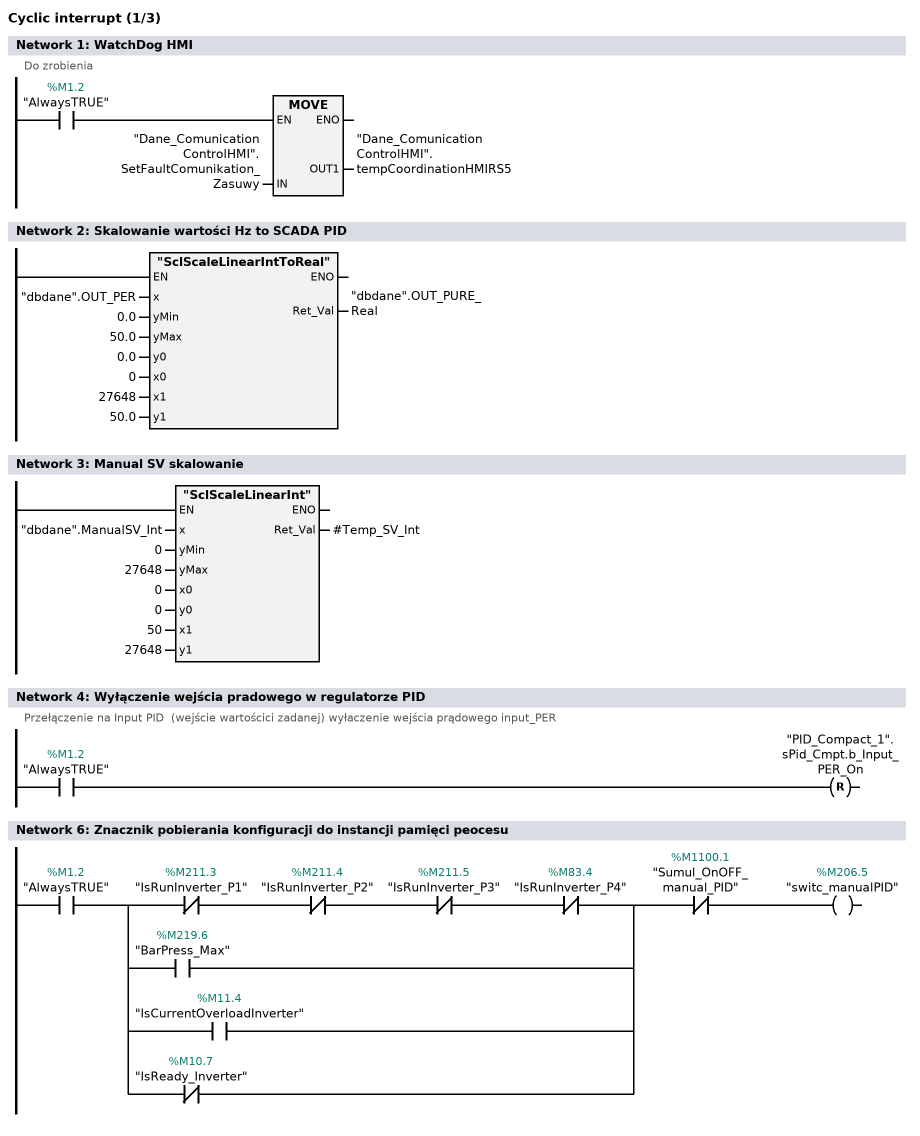
   RUNG wire#powerrail
      Contact( "AlwaysTRUE" )
      Move(in := "Dane_ComunicationControlHMI".SetFaultComunikation_Zasuwy, out1 => "Dane_ComunicationControlHMI".tempCoordinationHMIRS5)
   END_RUNG
   // the same network as SCL:
   IF "AlwaysTRUE" THEN
       "Dane_ComunicationControlHMI".tempCoordinationHMIRS5 := "Dane_ComunicationControlHMI".SetFaultComunikation_Zasuwy;
   END_IF;
END_REGION

REGION Network 2: Skalowanie wartości Hz to SCADA PID
   RUNG wire#powerrail
      "SclScaleLinearIntToReal"(x := "dbdane".OUT_PER, yMin := 0.0, yMax := 50.0, y0 := 0.0, x0 := 0, x1 := 27648, y1 := 50.0, Ret_Val => "dbdane".OUT_PURE_Real)
   END_RUNG
   // the same network as SCL:
   "dbdane".OUT_PURE_Real := "SclScaleLinearIntToReal"(x := "dbdane".OUT_PER,
                           yMin := 0.0,
                           yMax := 50.0,
                           y0 := 0.0,
                           x0 := 0,
                           x1 := 27648,
                           y1 := 50.0);
END_REGION

REGION Network 3: Manual SV skalowanie
   RUNG wire#powerrail
      "SclScaleLinearInt"(x := "dbdane".ManualSV_Int, yMin := 0, yMax := 27648, x0 := 0, y0 := 0, x1 := 50, y1 := 27648, Ret_Val => #Temp_SV_Int)
   END_RUNG
   // the same network as SCL:
   #Temp_SV_Int := "SclScaleLinearInt"(x := "dbdane".ManualSV_Int,
                           yMin := 0,
                           yMax := 27648,
                           x0 := 0,
                           y0 := 0,
                           x1 := 50,
                           y1 := 27648);
END_REGION

REGION Network 4: Wyłączenie wejścia pradowego w regulatorze PID
   // Przełączenie na Input PID  (wejście wartościci zadanej) wyłaczenie wejścia prądowego input_PER
   RUNG wire#powerrail
      Contact( "AlwaysTRUE" )
      R_Coil( "PID_Compact_1".sPid_Cmpt.b_Input_PER_On )
   END_RUNG
   // the same network as SCL:
   IF "AlwaysTRUE" THEN "PID_Compact_1".sPid_Cmpt.b_Input_PER_On := FALSE; END_IF;
END_REGION

REGION Network 5: Skalowanie wartośc pressure oxygen
   // Przetwornik ciśnienia (0-1bar) 
   // !!!!!! Znienić po zamontowaniu właściwego !!!!!!! 
   // obecnie czujnik 10 bar
END_REGION

REGION Network 6: Znacznik pobierania konfiguracji do instancji pamięci peocesu
   RUNG wire#powerrail
      Contact( "AlwaysTRUE" )
      wire#w1
      I_Contact( "IsRunInverter_P1" )
      I_Contact( "IsRunInverter_P2" )
      I_Contact( "IsRunInverter_P3" )
      I_Contact( "IsRunInverter_P4" )
      wire#w2
      I_Contact( "Sumul_OnOFF_manual_PID" )
      Coil( "switc_manualPID" )
   END_RUNG
   RUNG wire#w1
      Contact( "BarPress_Max" )
   END_RUNG wire#w2
   RUNG wire#w1
      Contact( "IsCurrentOverloadInverter" )
   END_RUNG wire#w2
   RUNG wire#w1
      I_Contact( "IsReady_Inverter" )
   END_RUNG wire#w2
   // the same network as SCL:
   "switc_manualPID" := "AlwaysTRUE" AND ((NOT "IsRunInverter_P1" AND NOT "IsRunInverter_P2" AND NOT "IsRunInverter_P3" AND NOT "IsRunInverter_P4") OR "BarPress_Max" OR "IsCurrentOverloadInverter" OR NOT "IsReady_Inverter") AND NOT "Sumul_OnOFF_manual_PID";
END_REGION

REGION Network 7: PID
   // Linia załączenia Manual wykonyje zadanie przekazania wartości minimalnej gdy nie pracuje falownik.
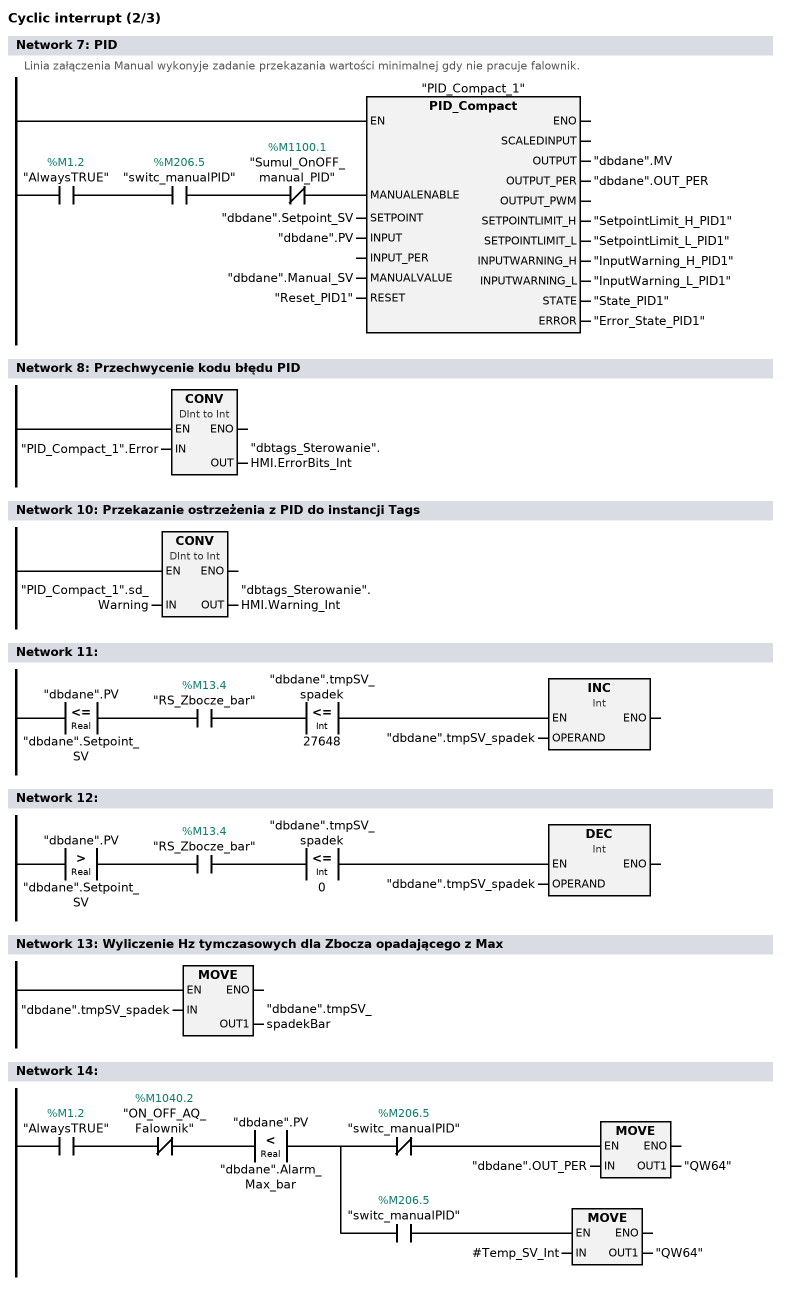
   RUNG wire#powerrail
      "PID_Compact_1".PID_Compact(ManualEnable := wire#w1, Setpoint := "dbdane".Setpoint_SV, Input := "dbdane".PV, Input_PER :=, ManualValue := "dbdane".Manual_SV, Reset := "Reset_PID1", ScaledInput =>, Output => "dbdane".MV, Output_PER => "dbdane".OUT_PER, Output_PWM =>, SetpointLimit_H => "SetpointLimit_H_PID1", SetpointLimit_L => "SetpointLimit_L_PID1", InputWarning_H => "InputWarning_H_PID1", InputWarning_L => "InputWarning_L_PID1", State => "State_PID1", Error => "Error_State_PID1")
   END_RUNG
   RUNG wire#powerrail
      Contact( "AlwaysTRUE" )
      Contact( "switc_manualPID" )
      I_Contact( "Sumul_OnOFF_manual_PID" )
   END_RUNG wire#w1
   // the same network as SCL:
   "PID_Compact_1"(ManualEnable := "AlwaysTRUE" AND "switc_manualPID" AND NOT "Sumul_OnOFF_manual_PID",   // PID_Compact
                   Setpoint := "dbdane".Setpoint_SV,
                   Input := "dbdane".PV,
                   ManualValue := "dbdane".Manual_SV,
                   Reset := "Reset_PID1",
                   Output => "dbdane".MV,
                   Output_PER => "dbdane".OUT_PER,
                   SetpointLimit_H => "SetpointLimit_H_PID1",
                   SetpointLimit_L => "SetpointLimit_L_PID1",
                   InputWarning_H => "InputWarning_H_PID1",
                   InputWarning_L => "InputWarning_L_PID1",
                   State => "State_PID1",
                   Error => "Error_State_PID1");
END_REGION

REGION Network 8: Przechwycenie kodu błędu PID
   RUNG wire#powerrail
      { S7_Templates := "[SrcType := DInt, DestType := Int]"; S7_GenerateENO := "TRUE" } Convert(in := "PID_Compact_1".Error, out => "dbtags_Sterowanie".HMI.ErrorBits_Int)
   END_RUNG
   // the same network as SCL:
   "dbtags_Sterowanie".HMI.ErrorBits_Int := DINT_TO_INT("PID_Compact_1".Error);
END_REGION

REGION Network 10: Przekazanie ostrzeżenia z PID do instancji Tags
   RUNG wire#powerrail
      { S7_Templates := "[SrcType := DInt, DestType := Int]"; S7_GenerateENO := "TRUE" } Convert(in := "PID_Compact_1".sd_Warning, out => "dbtags_Sterowanie".HMI.Warning_Int)
   END_RUNG
   // the same network as SCL:
   "dbtags_Sterowanie".HMI.Warning_Int := DINT_TO_INT("PID_Compact_1".sd_Warning);
END_REGION

REGION Network 11
   RUNG wire#powerrail
      { S7_Templates := "SrcType := Real" } LE_Contact(in1 := "dbdane".PV, in2 := "dbdane".Setpoint_SV)
      Contact( "RS_Zbocze_bar" )
      { S7_Templates := "SrcType := Int" } LE_Contact(in1 := "dbdane".tmpSV_spadek, in2 := 27648)
      { S7_Templates := "DestType := Int" } Inc( "dbdane".tmpSV_spadek )
   END_RUNG
   // the same network as SCL:
   IF ("dbdane".PV <= "dbdane".Setpoint_SV) AND "RS_Zbocze_bar" AND ("dbdane".tmpSV_spadek <= 27648) THEN
       "dbdane".tmpSV_spadek := "dbdane".tmpSV_spadek + 1;
   END_IF;
END_REGION

REGION Network 12
   RUNG wire#powerrail
      { S7_Templates := "SrcType := Real" } GT_Contact(in1 := "dbdane".PV, in2 := "dbdane".Setpoint_SV)
      Contact( "RS_Zbocze_bar" )
      { S7_Templates := "SrcType := Int" } LE_Contact(in1 := "dbdane".tmpSV_spadek, in2 := 0)
      { S7_Templates := "DestType := Int" } Dec( "dbdane".tmpSV_spadek )
   END_RUNG
   // the same network as SCL:
   IF ("dbdane".PV > "dbdane".Setpoint_SV) AND "RS_Zbocze_bar" AND ("dbdane".tmpSV_spadek <= 0) THEN
       "dbdane".tmpSV_spadek := "dbdane".tmpSV_spadek - 1;
   END_IF;
END_REGION

REGION Network 13: Wyliczenie Hz tymczasowych dla Zbocza opadającego z Max
   RUNG wire#powerrail
      Move(in := "dbdane".tmpSV_spadek, out1 => "dbdane".tmpSV_spadekBar)
   END_RUNG
   // the same network as SCL:
   "dbdane".tmpSV_spadekBar := "dbdane".tmpSV_spadek;
END_REGION

REGION Network 14
   RUNG wire#powerrail
      Contact( "AlwaysTRUE" )
      I_Contact( "ON_OFF_AQ_Falownik" )
      { S7_Templates := "SrcType := Real" } LT_Contact(in1 := "dbdane".PV, in2 := "dbdane".Alarm_Max_bar)
      wire#w1
      I_Contact( "switc_manualPID" )
      { S7_GenerateENO := "TRUE" } Move(in := "dbdane".OUT_PER, out1 => "QW64")
   END_RUNG
   RUNG wire#w1
      Contact( "switc_manualPID" )
      { S7_GenerateENO := "TRUE" } Move(in := #Temp_SV_Int, out1 => "QW64")
   END_RUNG
   // the same network as SCL:
   #_w1 := "AlwaysTRUE" AND NOT "ON_OFF_AQ_Falownik" AND ("dbdane".PV < "dbdane".Alarm_Max_bar);
   IF #_w1 AND NOT "switc_manualPID" THEN "QW64" := "dbdane".OUT_PER; END_IF;
   IF #_w1 AND "switc_manualPID" THEN "QW64" := #Temp_SV_Int; END_IF;
END_REGION

REGION Network 15: Wyłączenie regulacji Hz
   // Jeśli ciśnienie alarmowe ustawienie na wyjściu Hz = 0
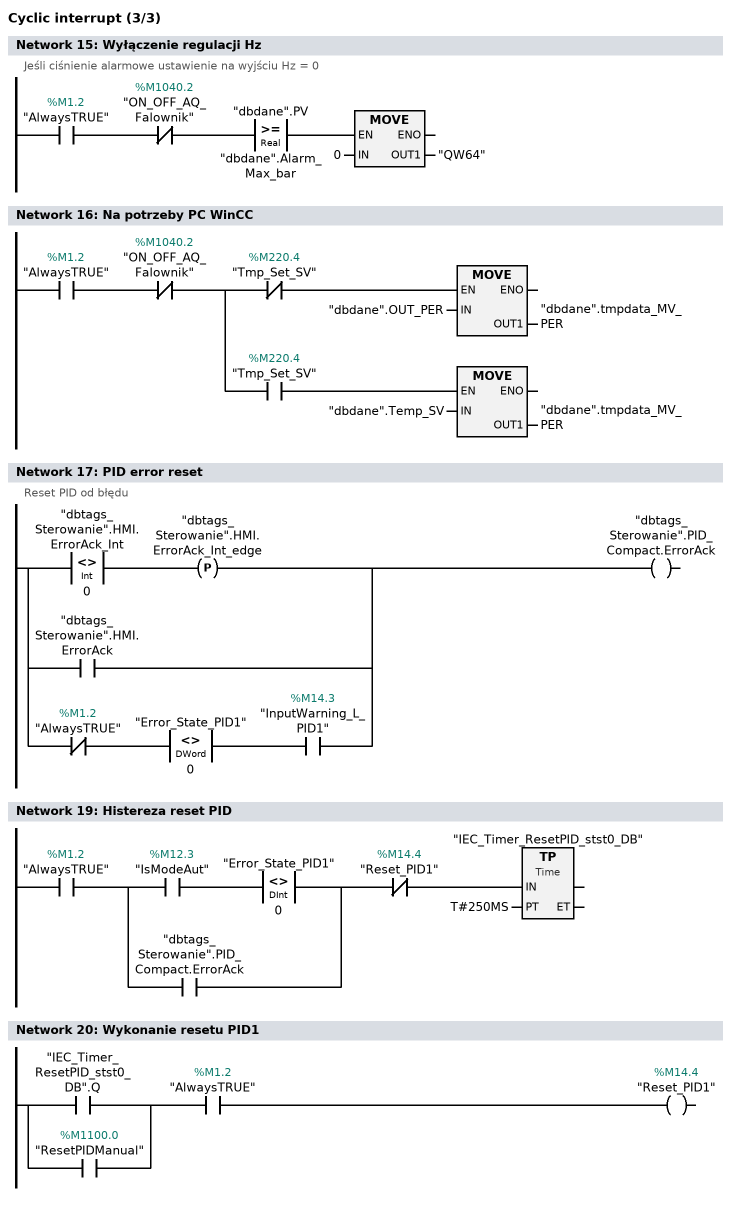
   RUNG wire#powerrail
      Contact( "AlwaysTRUE" )
      I_Contact( "ON_OFF_AQ_Falownik" )
      { S7_Templates := "SrcType := Real" } GE_Contact(in1 := "dbdane".PV, in2 := "dbdane".Alarm_Max_bar)
      { S7_GenerateENO := "TRUE" } Move(in := 0, out1 => "QW64")
   END_RUNG
   // the same network as SCL:
   IF "AlwaysTRUE" AND NOT "ON_OFF_AQ_Falownik" AND ("dbdane".PV >= "dbdane".Alarm_Max_bar) THEN
       "QW64" := 0;
   END_IF;
END_REGION

REGION Network 16: Na potrzeby PC WinCC
   RUNG wire#powerrail
      Contact( "AlwaysTRUE" )
      I_Contact( "ON_OFF_AQ_Falownik" )
      wire#w1
      I_Contact( "Tmp_Set_SV" )
      { S7_GenerateENO := "TRUE" } Move(in := "dbdane".OUT_PER, out1 => "dbdane".tmpdata_MV_PER)
   END_RUNG
   RUNG wire#w1
      Contact( "Tmp_Set_SV" )
      { S7_GenerateENO := "TRUE" } Move(in := "dbdane".Temp_SV, out1 => "dbdane".tmpdata_MV_PER)
   END_RUNG
   // the same network as SCL:
   #_w1 := "AlwaysTRUE" AND NOT "ON_OFF_AQ_Falownik";
   IF #_w1 AND NOT "Tmp_Set_SV" THEN "dbdane".tmpdata_MV_PER := "dbdane".OUT_PER; END_IF;
   IF #_w1 AND "Tmp_Set_SV" THEN "dbdane".tmpdata_MV_PER := "dbdane".Temp_SV; END_IF;
END_REGION

REGION Network 17: PID error reset
   // Reset PID od błędu
   RUNG wire#powerrail
      { S7_Templates := "SrcType := Int" } NE_Contact(in1 := "dbtags_Sterowanie".HMI.ErrorAck_Int, in2 := 0)
      P_Trig( "dbtags_Sterowanie".HMI.ErrorAck_Int_edge )
      wire#w1
      Coil( "dbtags_Sterowanie".PID_Compact.ErrorAck )
   END_RUNG
   RUNG wire#powerrail
      Contact( "dbtags_Sterowanie".HMI.ErrorAck )
   END_RUNG wire#w1
   RUNG wire#powerrail
      I_Contact( "AlwaysTRUE" )
      { S7_Templates := "SrcType := DWord" } NE_Contact(in1 := "Error_State_PID1", in2 := 0)
      Contact( "InputWarning_L_PID1" )
   END_RUNG wire#w1
   // the same network as SCL:
   #_w1 := "dbtags_Sterowanie".HMI.ErrorAck_Int <> 0;
   #_w2 := #_w1 AND NOT "dbtags_Sterowanie".HMI.ErrorAck_Int_edge;   // rising edge
   "dbtags_Sterowanie".HMI.ErrorAck_Int_edge := #_w1;
   "dbtags_Sterowanie".PID_Compact.ErrorAck := #_w2 OR "dbtags_Sterowanie".HMI.ErrorAck OR (NOT "AlwaysTRUE" AND ("Error_State_PID1" <> 0) AND "InputWarning_L_PID1");
END_REGION

REGION Network 19: Histereza reset PID
   RUNG wire#powerrail
      Contact( "AlwaysTRUE" )
      wire#w1
      Contact( "IsModeAut" )
      { S7_Templates := "SrcType := DInt" } NE_Contact(in1 := "Error_State_PID1", in2 := 0)
      wire#w2
      I_Contact( "Reset_PID1" )
      { S7_Templates := "time_type := Time" } "IEC_Timer_ResetPID_stst0_DB".TP(pt := T#250MS, et =>)
   END_RUNG
   RUNG wire#w1
      Contact( "dbtags_Sterowanie".PID_Compact.ErrorAck )
   END_RUNG wire#w2
   // the same network as SCL:
   "IEC_Timer_ResetPID_stst0_DB".TP(IN := "AlwaysTRUE" AND (("IsModeAut" AND ("Error_State_PID1" <> 0)) OR "dbtags_Sterowanie".PID_Compact.ErrorAck) AND NOT "Reset_PID1",
                           PT := T#250MS);
END_REGION

REGION Network 20: Wykonanie resetu PID1
   RUNG wire#powerrail
      Contact( "IEC_Timer_ResetPID_stst0_DB".Q )
      wire#w1
      Contact( "AlwaysTRUE" )
      Coil( "Reset_PID1" )
   END_RUNG
   RUNG wire#powerrail
      Contact( "ResetPIDManual" )
   END_RUNG wire#w1
   // the same network as SCL:
   "Reset_PID1" := ("IEC_Timer_ResetPID_stst0_DB".Q OR "ResetPIDManual") AND "AlwaysTRUE";
END_REGION
END_ORGANIZATION_BLOCK

ORGANIZATION_BLOCK "Cyclic interrupt_2"   // OB32, LAD, CyclicInterrupt
TITLE = Pobranie analogów z wejścia
{ S7_Optimized_Access := 'TRUE' }
AUTHOR : rtecmer
VERSION : 0.1
// Obsługa wejść analogowych
// stored: AutoNumber true, IsIECCheckEnabled false, SetENOAutomatically false
   VAR_INPUT
      Initial_Call : Bool;   // Initial call of this OB
      Event_Count : Int;   // Events discarded
   END_VAR
BEGIN

REGION Network 1: Pobranie wartości z wejść analogowych
   // B6 - Miasto
   // B7 - Pompownia
   // B8 - Suchobieg
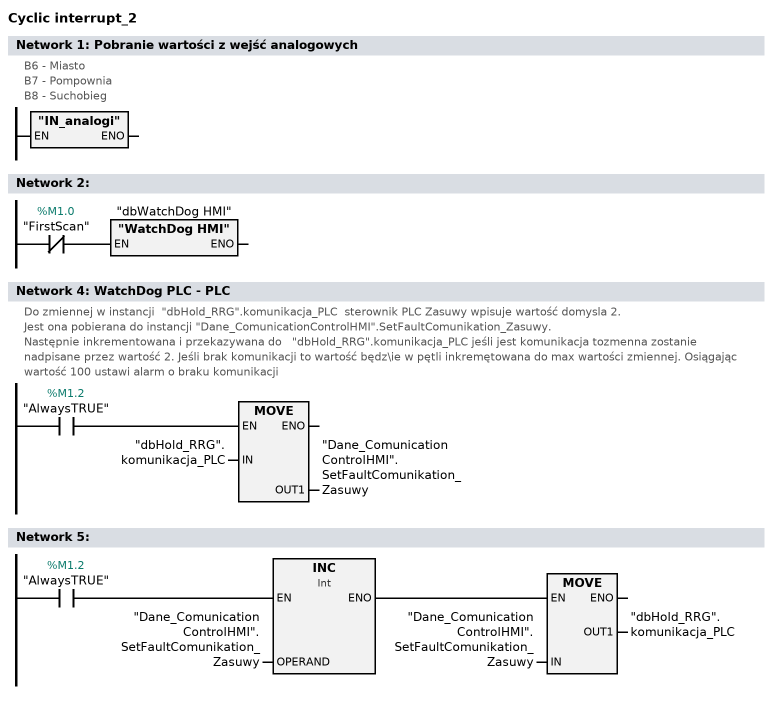
   RUNG wire#powerrail
      "IN_analogi"()
   END_RUNG
   // the same network as SCL:
   "IN_analogi"();
END_REGION

REGION Network 2
   RUNG wire#powerrail
      I_Contact( "FirstScan" )
      "dbWatchDog HMI"()
   END_RUNG
   // the same network as SCL:
   IF NOT "FirstScan" THEN
       "dbWatchDog HMI"();   // "WatchDog HMI"
   END_IF;
END_REGION

REGION Network 4: WatchDog PLC - PLC
   // Do zmiennej w instancji  "dbHold_RRG".komunikacja_PLC  sterownik PLC Zasuwy wpisuje wartość domysla 2.
   // Jest ona pobierana do instancji "Dane_ComunicationControlHMI".SetFaultComunikation_Zasuwy.
   // Następnie inkrementowana i przekazywana do   "dbHold_RRG".komunikacja_PLC jeśli jest komunikacja tozmenna zostanie nadpisane przez wartość 2. Jeśli brak komunikacji to wartość będz\ie w pętli inkremętowana do max wartości zmiennej. Osiągając wartość 100 ustawi alarm o braku komunikacji
   RUNG wire#powerrail
      Contact( "AlwaysTRUE" )
      Move(in := "dbHold_RRG".komunikacja_PLC, out1 => "Dane_ComunicationControlHMI".SetFaultComunikation_Zasuwy)
   END_RUNG
   // the same network as SCL:
   IF "AlwaysTRUE" THEN
       "Dane_ComunicationControlHMI".SetFaultComunikation_Zasuwy := "dbHold_RRG".komunikacja_PLC;
   END_IF;
END_REGION

REGION Network 5
   RUNG wire#powerrail
      Contact( "AlwaysTRUE" )
      { S7_Templates := "DestType := Int" } Inc( "Dane_ComunicationControlHMI".SetFaultComunikation_Zasuwy )
      Move(in := "Dane_ComunicationControlHMI".SetFaultComunikation_Zasuwy, out1 => "dbHold_RRG".komunikacja_PLC)
   END_RUNG
   // the same network as SCL:
   IF "AlwaysTRUE" THEN
       "Dane_ComunicationControlHMI".SetFaultComunikation_Zasuwy := "Dane_ComunicationControlHMI".SetFaultComunikation_Zasuwy + 1;
       "dbHold_RRG".komunikacja_PLC := "Dane_ComunicationControlHMI".SetFaultComunikation_Zasuwy;
   END_IF;
END_REGION

REGION Network 7 (SCL): Reset znaczników zbocza wysyłania danych przez TCP
   "memRisingTriger_Data_1" := FALSE;
   "memTrig_Client_Receiving_1" := FALSE;
   "memRisingTriger_Data_2" := FALSE;
   "memTrig_Client_Receiving_2" := FALSE;
   "memRisingTriger_Data_3" := FALSE;
   "memTrig_Client_Receiving_3" := FALSE;
   "memRisingTriger_Data_4" := FALSE;
   "memTrig_Client_Receiving_4" := FALSE;
   "memRisingTriger_Data_5" := FALSE;
   "memTrig_Client_Receiving_5" := FALSE;
   "memRisingTriger_Data_6" := FALSE;
   "memTrig_Client_Receiving_6" := FALSE;
   "memRisingTriger_Data_7" := FALSE;
   "memTrig_Client_Receiving_7" := FALSE;
   "memRisingTriger_Data_8" := FALSE;
   "memTrig_Client_Receiving_8" := FALSE;
   "memRisingTriger_Data_9" := FALSE;
   "memTrig_Client_Receiving_9" := FALSE;
   "memRisingTriger_Data_10" := FALSE;
   "memTrig_Client_Receiving_10" := FALSE;
END_REGION

REGION Network 8 (SCL): pamieć zbocza narastającego przekazania danej do wysłania
   "memRisingTriger_Data_11" := FALSE;
   "memTrig_Client_Receiving_11" := FALSE;
   "memRisingTriger_Data_12" := FALSE;
   "memTrig_Client_Receiving_12" := FALSE;
   "memRisingTriger_Data_13" := FALSE;
   "memTrig_Client_Receiving_13" := FALSE;
   "memRisingTriger_Data_14" := FALSE;
   "memTrig_Client_Receiving_14" := FALSE;
   "memRisingTriger_Data_15" := FALSE;
   "memTrig_Client_Receiving_15" := FALSE;
   "memRisingTriger_Data_16" := FALSE;
   "memTrig_Client_Receiving_16" := FALSE;
   "memRisingTriger_Data_17" := FALSE;
   "memTrig_Client_Receiving_17" := FALSE;
   "memRisingTriger_Data_18" := FALSE;
   "memTrig_Client_Receiving_18" := FALSE;
   "memRisingTriger_Data_19" := FALSE;
   "memTrig_Client_Receiving_19" := FALSE;
   "memRisingTriger_Data_20" := FALSE;
   "memTrig_Client_Receiving_20" := FALSE;
END_REGION
END_ORGANIZATION_BLOCK

FUNCTION "IN_analogi" : Void
TITLE = Przekazanie wartości z wejść analogowych
{ S7_Optimized_Access := 'TRUE' }
AUTHOR : rtecmer
VERSION : 0.1
//(*
////=============================================================================
////(JZWiK S.A Radosław Tecmer)
////(c)Copyright (2021) All Rights Reserved
////-----------------------------------------------------------------------------
////Testowane z:   (system docelowy z  FW 4.4)
////Pakiet inżynierski:   TIA Portal (V14 Sp1 Update 9)
////Ograniczenia:  ( - )
////Wymagania:  (minimalne S7-1200 CPU 1215C FW 4.2 .)
////Funkcjonalnośc: (Pobranie wartości z wejść analogowych )
////-----------------------------------------------------------------------------
////Zmainy wprowadzone:
////Wersja  Data       Osoba wprowadzająca zmiany - ekspert
////01.00.00 11.01.2022 (Tecmer Radosław - twórca) Pieresza wersja 01.00.00
////=============================================================================
//*)

BEGIN
	(*
	//=============================================================================
	//(JZWiK S.A Radosław Tecmer)
	//(c)Copyright (2021) All Rights Reserved
	//-----------------------------------------------------------------------------
	//Testowane z:   (system docelowy z  FW 4.4)
	//Pakiet inżynierski:   TIA Portal (V14 Sp1 Update 9)
	//Ograniczenia:  ( - )
	//Wymagania:  (minimalne S7-1200 CPU 1215C FW 4.2 .)
	//Funkcjonalnośc: (Pobranie wartości z wejść analogowych )
	//-----------------------------------------------------------------------------
	//Zmainy wprowadzone:
	//Wersja  Data       Osoba wprowadzająca zmiany - ekspert
	//01.00.00 11.01.2022 (Tecmer Radosław - twórca) Pieresza wersja 01.00.00
	//=============================================================================
	*)
	
	// ciśnienie przetłaczania miasto
	IF "dbdane".PV_analaog_B6 > 0.2 THEN // czy nie uszkodzone rury
	  IF "dbdane".PV_analaog_B6 < 27651 THEN // przerwana pętla prądowa
	    // to przekazanie wartości
	    "dbdane".PV_PER_B6 := "dbdane".PV_analaog_B6;
	  ELSE
	    "dbdane".PV_PER_B6 := 32767;
	    ;
	  END_IF;
	  
	  ;
	END_IF;
	
	
	
	// ciśnienie pompownia
	IF "dbdane".PV_analaog_B7 > 0.2 THEN // czy nie uszkodzone rury
	  IF "dbdane".PV_analaog_B7 < 27651 THEN // przerwana pętla prądowa
	    // to przekazanie wartości
	    "dbdane".PV_PER_B7 := "dbdane".PV_analaog_B7;
	    ;
	  ELSE
	    "dbdane".PV_PER_B7 := 32767;
	    ;
	  END_IF;
	  
	  ;
	END_IF;
	
	
	//ciśnienie ssania
	IF  "dbdane".PV_analaog_B8 > 0.2 THEN // czy nie uszkodzone rury
	  // to przekazanie wartości
	  "dbdane".PV_PER_B8 := "dbdane".PV_analaog_B8;
	ELSE
	  "dbdane".PV_PER_B8 := 0;
	  ;
	END_IF;
	
	
	
	
	// przepływ analog
	"dbdane".actPrzepływQ1_IA := "IW70":P;
	
	"dbdane".actPrzepływQ1_IA_real := "SclScaleLinearIntToReal"(x := "dbdane".actPrzepływQ1_IA, yMin := 0.0, yMax := 600.0, y0 := 0.0, x0 := 0, x1 := 27648, y1 := 600.0);
	
END_FUNCTION

FUNCTION_BLOCK "WatchDog HMI"   // FB12, LAD
TITLE = WatchDog HMI
{ S7_Optimized_Access := 'TRUE' }
AUTHOR : rtecmer
VERSION : 0.1
// Kontrola komunikacji PLC z HMI.  Wartość w zmiennej w instancji "Dane_ComunicationControlHMI".tempCoordinationHMIRS5 jest inkrementowana przez PLC i co minutę skrypt z HMI wartość zeruje. Jeśli błąd kumunikacj to wartość jest inkrementowana do max zmiennej. Przy wartości 70 ustawiany jest bit alarmu dla PLC, że btrak komunikacji z HMI
// HMI na podstawie błędu systemowego 190011 komonikuje w tabeli alarmów o braku komunikacji
// stored: AutoNumber true, IsIECCheckEnabled false, IsRetainMemResEnabled false, MemoryReserve 500, SetENOAutomatically false, UDAEnableTagReadback false
   VAR_TEMP   // added for the SCL form of the ladder/FBD networks
      _w1 : Bool;
      _w2 : Bool;
   END_VAR
BEGIN

REGION Network 1: WatchDog HMI
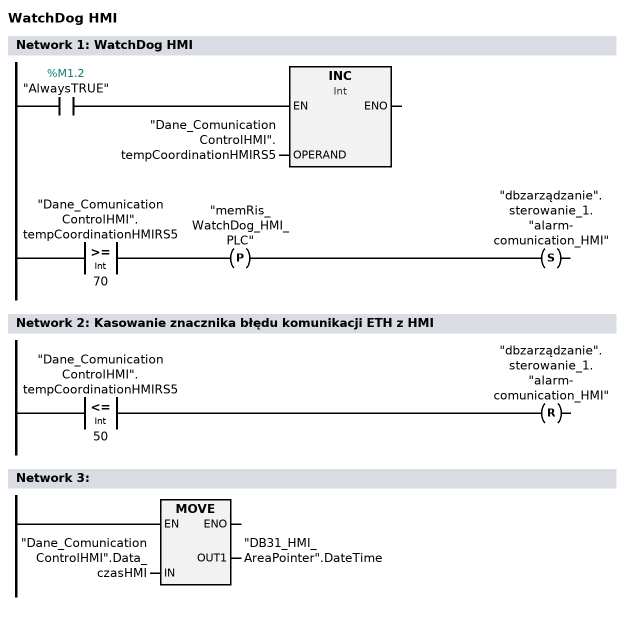
   RUNG wire#powerrail
      Contact( "AlwaysTRUE" )
      { S7_Templates := "DestType := Int" } Inc( "Dane_ComunicationControlHMI".tempCoordinationHMIRS5 )
   END_RUNG
   RUNG wire#powerrail
      { S7_Templates := "SrcType := Int" } GE_Contact(in1 := "Dane_ComunicationControlHMI".tempCoordinationHMIRS5, in2 := 70)
      P_Trig( "memRis_WatchDog_HMI_PLC" )
      S_Coil( "dbzarządzanie".sterowanie_1."alarm-comunication_HMI" )
   END_RUNG
   // the same network as SCL:
   IF "AlwaysTRUE" THEN
       "Dane_ComunicationControlHMI".tempCoordinationHMIRS5 := "Dane_ComunicationControlHMI".tempCoordinationHMIRS5 + 1;
   END_IF;
   #_w1 := "Dane_ComunicationControlHMI".tempCoordinationHMIRS5 >= 70;
   #_w2 := #_w1 AND NOT "memRis_WatchDog_HMI_PLC";   // rising edge
   "memRis_WatchDog_HMI_PLC" := #_w1;
   IF #_w2 THEN "dbzarządzanie".sterowanie_1."alarm-comunication_HMI" := TRUE; END_IF;
END_REGION

REGION Network 2: Kasowanie znacznika błędu komunikacji ETH z HMI
   RUNG wire#powerrail
      { S7_Templates := "SrcType := Int" } LE_Contact(in1 := "Dane_ComunicationControlHMI".tempCoordinationHMIRS5, in2 := 50)
      R_Coil( "dbzarządzanie".sterowanie_1."alarm-comunication_HMI" )
   END_RUNG
   // the same network as SCL:
   IF "Dane_ComunicationControlHMI".tempCoordinationHMIRS5 <= 50 THEN
       "dbzarządzanie".sterowanie_1."alarm-comunication_HMI" := FALSE;
   END_IF;
END_REGION

REGION Network 3
   RUNG wire#powerrail
      Move(in := "Dane_ComunicationControlHMI".Data_czasHMI, out1 => "DB31_HMI_AreaPointer".DateTime)
   END_RUNG
   // the same network as SCL:
   "DB31_HMI_AreaPointer".DateTime := "Dane_ComunicationControlHMI".Data_czasHMI;
END_REGION
END_FUNCTION_BLOCK

ORGANIZATION_BLOCK "Cyclic interrupt_SlaveModbusRTU"   // OB31, LAD, CyclicInterrupt
TITLE = Slave Modbus RTU
{ S7_Optimized_Access := 'TRUE' }
AUTHOR : rtecmer
VERSION : 0.1
// stored: AutoNumber true, IsIECCheckEnabled false, SetENOAutomatically false
   VAR_INPUT
      Initial_Call : Bool;   // Initial call of this OB
      Event_Count : Int;   // Events discarded
   END_VAR
BEGIN

REGION Network 1: ustawienie adresu slave PLC
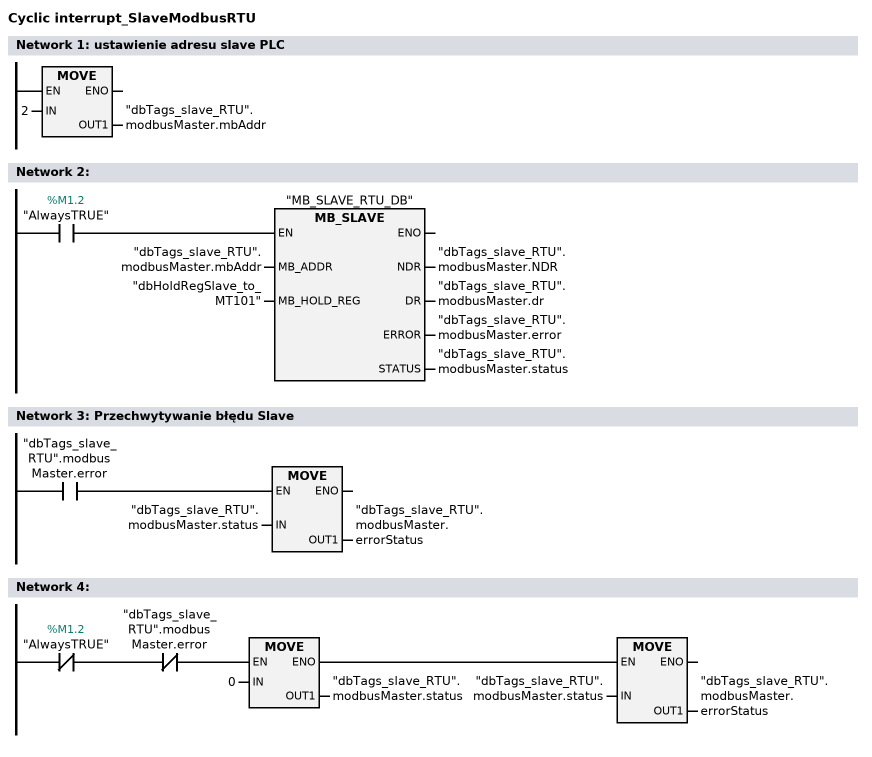
   RUNG wire#powerrail
      Move(in := 2, out1 => "dbTags_slave_RTU".modbusMaster.mbAddr)
   END_RUNG
   // the same network as SCL:
   "dbTags_slave_RTU".modbusMaster.mbAddr := 2;
END_REGION

REGION Network 2
   RUNG wire#powerrail
      Contact( "AlwaysTRUE" )
      "MB_SLAVE_RTU_DB".MB_SLAVE(MB_ADDR := "dbTags_slave_RTU".modbusMaster.mbAddr, MB_HOLD_REG := "dbHoldRegSlave_to_MT101", NDR => "dbTags_slave_RTU".modbusMaster.NDR, DR => "dbTags_slave_RTU".modbusMaster.dr, ERROR => "dbTags_slave_RTU".modbusMaster.error, STATUS => "dbTags_slave_RTU".modbusMaster.status)
   END_RUNG
   // the same network as SCL:
   IF "AlwaysTRUE" THEN
       "MB_SLAVE_RTU_DB"(MB_ADDR := "dbTags_slave_RTU".modbusMaster.mbAddr,   // MB_SLAVE
                         MB_HOLD_REG := "dbHoldRegSlave_to_MT101",
                         NDR => "dbTags_slave_RTU".modbusMaster.NDR,
                         DR => "dbTags_slave_RTU".modbusMaster.dr,
                         ERROR => "dbTags_slave_RTU".modbusMaster.error,
                         STATUS => "dbTags_slave_RTU".modbusMaster.status);
   END_IF;
END_REGION

REGION Network 3: Przechwytywanie błędu Slave
   RUNG wire#powerrail
      Contact( "dbTags_slave_RTU".modbusMaster.error )
      Move(in := "dbTags_slave_RTU".modbusMaster.status, out1 => "dbTags_slave_RTU".modbusMaster.errorStatus)
   END_RUNG
   // the same network as SCL:
   IF "dbTags_slave_RTU".modbusMaster.error THEN
       "dbTags_slave_RTU".modbusMaster.errorStatus := "dbTags_slave_RTU".modbusMaster.status;
   END_IF;
END_REGION

REGION Network 4
   RUNG wire#powerrail
      I_Contact( "AlwaysTRUE" )
      I_Contact( "dbTags_slave_RTU".modbusMaster.error )
      Move(in := 0, out1 => "dbTags_slave_RTU".modbusMaster.status)
      Move(in := "dbTags_slave_RTU".modbusMaster.status, out1 => "dbTags_slave_RTU".modbusMaster.errorStatus)
   END_RUNG
   // the same network as SCL:
   IF NOT "AlwaysTRUE" AND NOT "dbTags_slave_RTU".modbusMaster.error THEN
       "dbTags_slave_RTU".modbusMaster.status := 0;
       "dbTags_slave_RTU".modbusMaster.errorStatus := "dbTags_slave_RTU".modbusMaster.status;
   END_IF;
END_REGION
END_ORGANIZATION_BLOCK

ORGANIZATION_BLOCK "Diagnostic error interrupt"   // OB82, LAD, DiagnosticErrorInterrupt
TITLE = Diagnostyka błedów
{ S7_Optimized_Access := 'TRUE' }
AUTHOR : rtecmer
VERSION : 0.1
// stored: IsIECCheckEnabled false, SetENOAutomatically false
   VAR_INPUT
      IO_State : Word;   // IO state of the HW object
      LADDR : HW_ANY;   // Hardware identifier
      Channel : UInt;   // Channel number
      MultiError : Bool;   // =true if more than one error is present
   END_VAR
   VAR_TEMP
      RetVal_RD_SYS_T : Int;   // //Status of the instruction RD_SYS_T: Read time-of-day
   END_VAR
BEGIN

REGION Network 2 (SCL)
   "EX012_ErrorBuffer_OB82".OB82ErrorCounter := "EX012_ErrorBuffer_OB82".OB82ErrorCounter + 1;
   //ochrona przed przepełnieniem tabeli
   IF ("EX012_ErrorBuffer_OB82".OB82ErrorCounter > "CONST_BUFFER_OB82") THEN
     "EX012_ErrorBuffer_OB82".OB82ErrorCounter := 1;
   END_IF;
   //Wystąpił błąd czasu
   #RetVal_RD_SYS_T := RD_LOC_T(OUT => "EX012_ErrorBuffer_OB82".ErrorDataOB82["EX012_ErrorBuffer_OB82".OB82ErrorCounter].ErrorTimestamp);
   //Zapis błedu do buffora (ErrorBuffor)
   "EX012_ErrorBuffer_OB82".ErrorDataOB82["EX012_ErrorBuffer_OB82".OB82ErrorCounter].IO_State := #IO_State;
   "EX012_ErrorBuffer_OB82".ErrorDataOB82["EX012_ErrorBuffer_OB82".OB82ErrorCounter].LADDR := #LADDR;
   "EX012_ErrorBuffer_OB82".ErrorDataOB82["EX012_ErrorBuffer_OB82".OB82ErrorCounter].Channel := #Channel;
   "EX012_ErrorBuffer_OB82".ErrorDataOB82["EX012_ErrorBuffer_OB82".OB82ErrorCounter].MultiError := #MultiError;
END_REGION
END_ORGANIZATION_BLOCK

ORGANIZATION_BLOCK "Hardware interrupt Reset"   // OB40, LAD, HardwareInterrupt
TITLE = Reset
{ S7_Optimized_Access := 'TRUE' }
AUTHOR : rtecmer
VERSION : 0.1
// Ustawienie gotowości i tryb
// stored: AutoNumber true, IsIECCheckEnabled false, SetENOAutomatically false
   VAR_INPUT
      LADDR : HW_IO;   // Hardware identifier
      USI : Word;   // User structure identifier
      IChannel : USInt;   // Interrupt channel number
      EventType : Byte;   // EventType
   END_VAR
BEGIN
END_ORGANIZATION_BLOCK

ORGANIZATION_BLOCK "Reset_falling_edge_PowerRS5"   // OB41, LAD, HardwareInterrupt
TITLE = Reset po braku zasilania RS5
{ S7_Optimized_Access := 'TRUE' }
AUTHOR : rtecmer
VERSION : 0.1
// Reset napędów po braku zasilania przy opadającym zboczu Power RS5
// stored: AutoNumber true, IsIECCheckEnabled false, SetENOAutomatically false
   VAR_INPUT
      LADDR : HW_IO;   // Hardware identifier
      USI : Word;   // User structure identifier
      IChannel : USInt;   // Interrupt channel number
      EventType : Byte;   // EventType
   END_VAR
BEGIN
END_ORGANIZATION_BLOCK

ORGANIZATION_BLOCK "Startup"   // OB100, LAD, Startup
TITLE = "Complete Restart"
{ S7_Optimized_Access := 'TRUE' }
AUTHOR : RTecmer
VERSION : 0.1
// stored: AutoNumber true, IsIECCheckEnabled false, SetENOAutomatically false
   VAR_INPUT
      LostRetentive : Bool;   // True if retentive data are lost
      LostRTC : Bool;   // True if date and time are lost
   END_VAR
BEGIN

REGION Network 1: inicjacja master modbus RTU / Incjalizacja modułu Master CM1241 (RS485) Modbus RTU
   // Komunikacja z przepływomierzami MP04 i falownikiem Danfoss
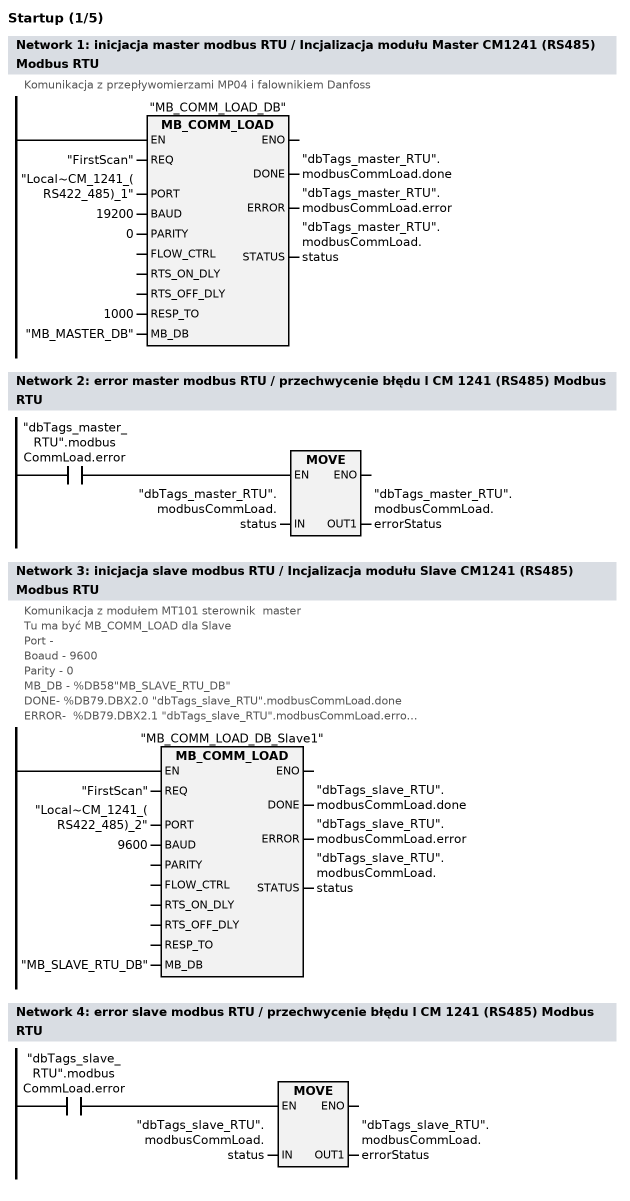
   RUNG wire#powerrail
      "MB_COMM_LOAD_DB".MB_COMM_LOAD(REQ := "FirstScan", PORT := "Local~CM_1241_(RS422_485)_1", BAUD := 19200, PARITY := 0, FLOW_CTRL :=, RTS_ON_DLY :=, RTS_OFF_DLY :=, RESP_TO := 1000, MB_DB := "MB_MASTER_DB", DONE => "dbTags_master_RTU".modbusCommLoad.done, ERROR => "dbTags_master_RTU".modbusCommLoad.error, STATUS => "dbTags_master_RTU".modbusCommLoad.status)
   END_RUNG
   // the same network as SCL:
   "MB_COMM_LOAD_DB"(REQ := "FirstScan",   // MB_COMM_LOAD
                     PORT := "Local~CM_1241_(RS422_485)_1",
                     BAUD := 19200,
                     PARITY := 0,
                     RESP_TO := 1000,
                     MB_DB := "MB_MASTER_DB",
                     DONE => "dbTags_master_RTU".modbusCommLoad.done,
                     ERROR => "dbTags_master_RTU".modbusCommLoad.error,
                     STATUS => "dbTags_master_RTU".modbusCommLoad.status);
END_REGION

REGION Network 2: error master modbus RTU / przechwycenie błędu l CM 1241 (RS485) Modbus RTU
   RUNG wire#powerrail
      Contact( "dbTags_master_RTU".modbusCommLoad.error )
      { S7_GenerateENO := "TRUE" } Move(in := "dbTags_master_RTU".modbusCommLoad.status, out1 => "dbTags_master_RTU".modbusCommLoad.errorStatus)
   END_RUNG
   // the same network as SCL:
   IF "dbTags_master_RTU".modbusCommLoad.error THEN
       "dbTags_master_RTU".modbusCommLoad.errorStatus := "dbTags_master_RTU".modbusCommLoad.status;
   END_IF;
END_REGION

REGION Network 3: inicjacja slave modbus RTU / Incjalizacja modułu Slave CM1241 (RS485) Modbus RTU
   // Komunikacja z modułem MT101 sterownik  master
   // 
   // Tu ma być MB_COMM_LOAD dla Slave
   // Port -
   // Boaud - 9600
   // Parity - 0
   // MB_DB - %DB58"MB_SLAVE_RTU_DB"
   // DONE- %DB79.DBX2.0 "dbTags_slave_RTU".modbusCommLoad.done
   // ERROR-  %DB79.DBX2.1 "dbTags_slave_RTU".modbusCommLoad.error
   // STATUS - %DB79.DBX2.2 "dbTags_slave_RTU".modbusCommLoad.status
   RUNG wire#powerrail
      "MB_COMM_LOAD_DB_Slave1".MB_COMM_LOAD(REQ := "FirstScan", PORT := "Local~CM_1241_(RS422_485)_2", BAUD := 9600, PARITY :=, FLOW_CTRL :=, RTS_ON_DLY :=, RTS_OFF_DLY :=, RESP_TO :=, MB_DB := "MB_SLAVE_RTU_DB", DONE => "dbTags_slave_RTU".modbusCommLoad.done, ERROR => "dbTags_slave_RTU".modbusCommLoad.error, STATUS => "dbTags_slave_RTU".modbusCommLoad.status)
   END_RUNG
   // the same network as SCL:
   "MB_COMM_LOAD_DB_Slave1"(REQ := "FirstScan",   // MB_COMM_LOAD
                           PORT := "Local~CM_1241_(RS422_485)_2",
                           BAUD := 9600,
                           MB_DB := "MB_SLAVE_RTU_DB",
                           DONE => "dbTags_slave_RTU".modbusCommLoad.done,
                           ERROR => "dbTags_slave_RTU".modbusCommLoad.error,
                           STATUS => "dbTags_slave_RTU".modbusCommLoad.status);
END_REGION

REGION Network 4: error slave modbus RTU / przechwycenie błędu l CM 1241 (RS485) Modbus RTU
   RUNG wire#powerrail
      Contact( "dbTags_slave_RTU".modbusCommLoad.error )
      { S7_GenerateENO := "TRUE" } Move(in := "dbTags_slave_RTU".modbusCommLoad.status, out1 => "dbTags_slave_RTU".modbusCommLoad.errorStatus)
   END_RUNG
   // the same network as SCL:
   IF "dbTags_slave_RTU".modbusCommLoad.error THEN
       "dbTags_slave_RTU".modbusCommLoad.errorStatus := "dbTags_slave_RTU".modbusCommLoad.status;
   END_IF;
END_REGION

REGION Network 5: Znacznik dodatkowej pompy dla funkcji FB8 I / Znacznik dodatkowego kompresora dla funkcji FB8 I
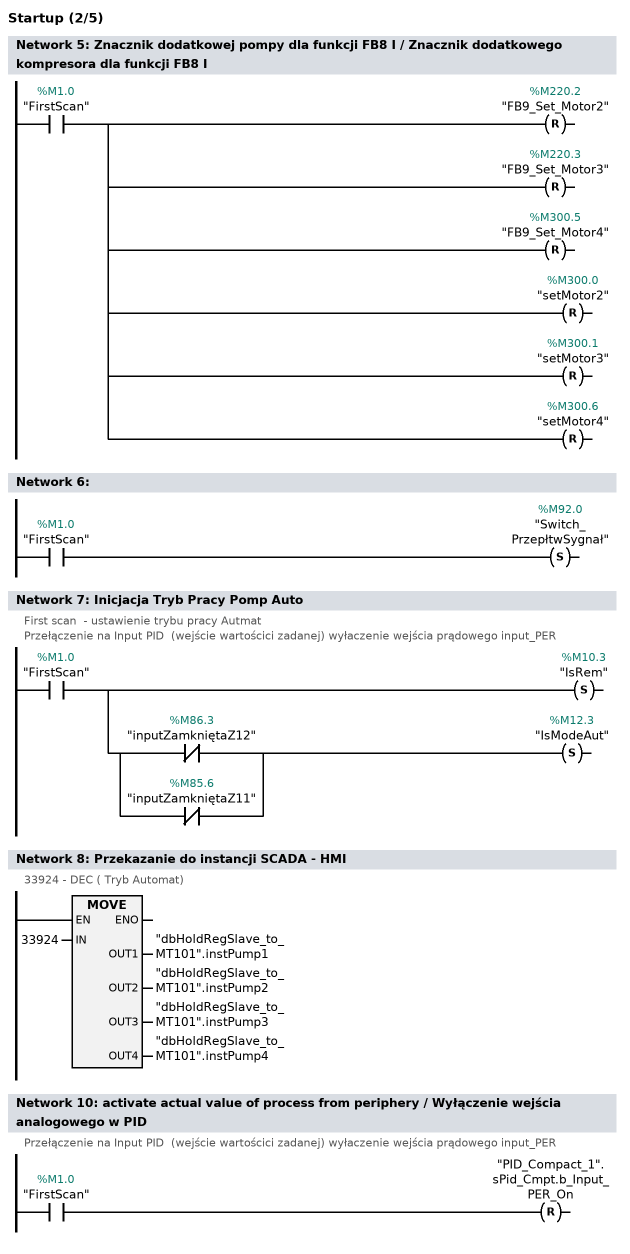
   RUNG wire#powerrail
      Contact( "FirstScan" )
      wire#w1
      R_Coil( "FB9_Set_Motor2" )
   END_RUNG
   RUNG wire#w1
      R_Coil( "FB9_Set_Motor3" )
   END_RUNG
   RUNG wire#w1
      R_Coil( "FB9_Set_Motor4" )
   END_RUNG
   RUNG wire#w1
      R_Coil( "setMotor2" )
   END_RUNG
   RUNG wire#w1
      R_Coil( "setMotor3" )
   END_RUNG
   RUNG wire#w1
      R_Coil( "setMotor4" )
   END_RUNG
   // the same network as SCL:
   IF "FirstScan" THEN
       "FB9_Set_Motor2" := FALSE;
       "FB9_Set_Motor3" := FALSE;
       "FB9_Set_Motor4" := FALSE;
       "setMotor2" := FALSE;
       "setMotor3" := FALSE;
       "setMotor4" := FALSE;
   END_IF;
END_REGION

REGION Network 6
   RUNG wire#powerrail
      Contact( "FirstScan" )
      S_Coil( "Switch_PrzepłtwSygnał" )
   END_RUNG
   // the same network as SCL:
   IF "FirstScan" THEN "Switch_PrzepłtwSygnał" := TRUE; END_IF;
END_REGION

REGION Network 7: Inicjacja Tryb Pracy Pomp Auto
   // First scan  - ustawienie trybu pracy Autmat 
   // Przełączenie na Input PID  (wejście wartościci zadanej) wyłaczenie wejścia prądowego input_PER
   RUNG wire#powerrail
      Contact( "FirstScan" )
      wire#w1
      S_Coil( "IsRem" )
   END_RUNG
   RUNG wire#w1
      I_Contact( "inputZamkniętaZ12" )
      wire#w2
      S_Coil( "IsModeAut" )
   END_RUNG
   RUNG wire#w1
      I_Contact( "inputZamkniętaZ11" )
   END_RUNG wire#w2
   // the same network as SCL:
   IF "FirstScan" THEN "IsRem" := TRUE; END_IF;
   IF "FirstScan" AND (NOT "inputZamkniętaZ12" OR NOT "inputZamkniętaZ11") THEN "IsModeAut" := TRUE; END_IF;
END_REGION

REGION Network 8: Przekazanie do instancji SCADA - HMI
   // 33924 - DEC ( Tryb Automat)
   RUNG wire#powerrail
      { S7_GenerateENO := "TRUE" } Move(in := 33924, out1 => "dbHoldRegSlave_to_MT101".instPump1, out2 => "dbHoldRegSlave_to_MT101".instPump2, out3 => "dbHoldRegSlave_to_MT101".instPump3, out4 => "dbHoldRegSlave_to_MT101".instPump4)
   END_RUNG
   // the same network as SCL:
   "dbHoldRegSlave_to_MT101".instPump1 := 33924;
   "dbHoldRegSlave_to_MT101".instPump2 := 33924;
   "dbHoldRegSlave_to_MT101".instPump3 := 33924;
   "dbHoldRegSlave_to_MT101".instPump4 := 33924;
END_REGION

REGION Network 10: activate actual value of process from periphery / Wyłączenie wejścia analogowego w PID
   // Przełączenie na Input PID  (wejście wartościci zadanej) wyłaczenie wejścia prądowego input_PER
   RUNG wire#powerrail
      Contact( "FirstScan" )
      R_Coil( "PID_Compact_1".sPid_Cmpt.b_Input_PER_On )
   END_RUNG
   // the same network as SCL:
   IF "FirstScan" THEN "PID_Compact_1".sPid_Cmpt.b_Input_PER_On := FALSE; END_IF;
END_REGION

REGION Network 11: Przekazanie nastaw
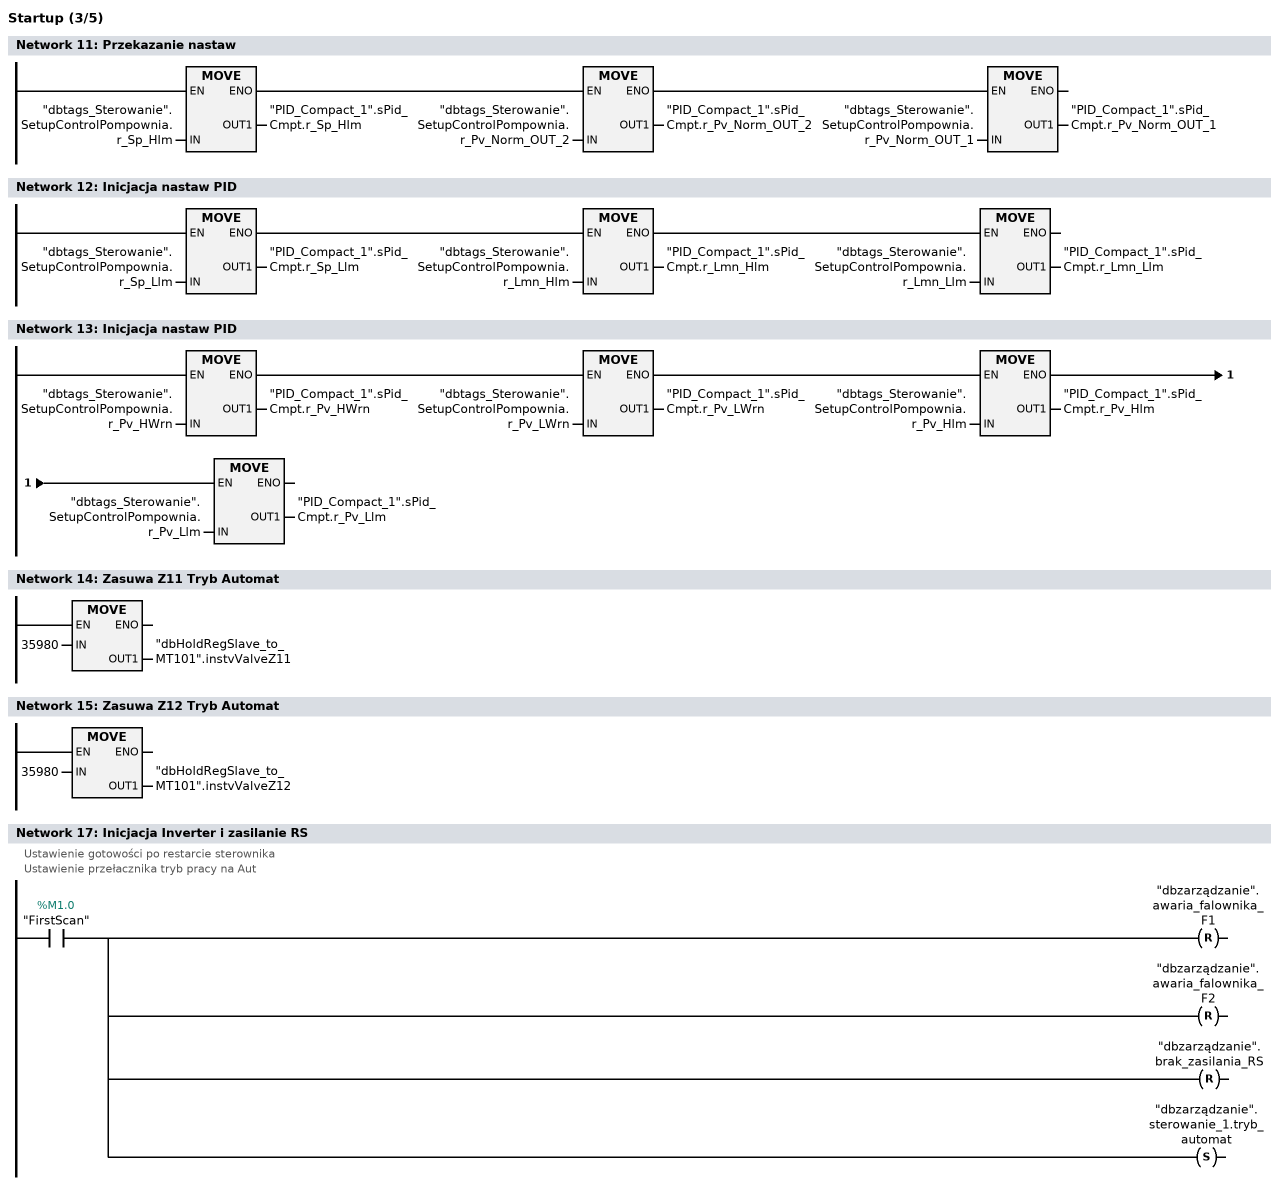
   RUNG wire#powerrail
      { S7_GenerateENO := "TRUE" } Move(in := "dbtags_Sterowanie".SetupControlPompownia.r_Sp_Hlm, out1 => "PID_Compact_1".sPid_Cmpt.r_Sp_Hlm)
      { S7_GenerateENO := "TRUE" } Move(in := "dbtags_Sterowanie".SetupControlPompownia.r_Pv_Norm_OUT_2, out1 => "PID_Compact_1".sPid_Cmpt.r_Pv_Norm_OUT_2)
      { S7_GenerateENO := "TRUE" } Move(in := "dbtags_Sterowanie".SetupControlPompownia.r_Pv_Norm_OUT_1, out1 => "PID_Compact_1".sPid_Cmpt.r_Pv_Norm_OUT_1)
   END_RUNG
   // the same network as SCL:
   // ENO of a box is taken as its EN; it also drops when the box reports an error
   "PID_Compact_1".sPid_Cmpt.r_Sp_Hlm := "dbtags_Sterowanie".SetupControlPompownia.r_Sp_Hlm;
   "PID_Compact_1".sPid_Cmpt.r_Pv_Norm_OUT_2 := "dbtags_Sterowanie".SetupControlPompownia.r_Pv_Norm_OUT_2;
   "PID_Compact_1".sPid_Cmpt.r_Pv_Norm_OUT_1 := "dbtags_Sterowanie".SetupControlPompownia.r_Pv_Norm_OUT_1;
END_REGION

REGION Network 12: Inicjacja nastaw PID
   RUNG wire#powerrail
      { S7_GenerateENO := "TRUE" } Move(in := "dbtags_Sterowanie".SetupControlPompownia.r_Sp_Llm, out1 => "PID_Compact_1".sPid_Cmpt.r_Sp_Llm)
      { S7_GenerateENO := "TRUE" } Move(in := "dbtags_Sterowanie".SetupControlPompownia.r_Lmn_Hlm, out1 => "PID_Compact_1".sPid_Cmpt.r_Lmn_Hlm)
      { S7_GenerateENO := "TRUE" } Move(in := "dbtags_Sterowanie".SetupControlPompownia.r_Lmn_Llm, out1 => "PID_Compact_1".sPid_Cmpt.r_Lmn_Llm)
   END_RUNG
   // the same network as SCL:
   // ENO of a box is taken as its EN; it also drops when the box reports an error
   "PID_Compact_1".sPid_Cmpt.r_Sp_Llm := "dbtags_Sterowanie".SetupControlPompownia.r_Sp_Llm;
   "PID_Compact_1".sPid_Cmpt.r_Lmn_Hlm := "dbtags_Sterowanie".SetupControlPompownia.r_Lmn_Hlm;
   "PID_Compact_1".sPid_Cmpt.r_Lmn_Llm := "dbtags_Sterowanie".SetupControlPompownia.r_Lmn_Llm;
END_REGION

REGION Network 13: Inicjacja nastaw PID
   RUNG wire#powerrail
      { S7_GenerateENO := "TRUE" } Move(in := "dbtags_Sterowanie".SetupControlPompownia.r_Pv_HWrn, out1 => "PID_Compact_1".sPid_Cmpt.r_Pv_HWrn)
      { S7_GenerateENO := "TRUE" } Move(in := "dbtags_Sterowanie".SetupControlPompownia.r_Pv_LWrn, out1 => "PID_Compact_1".sPid_Cmpt.r_Pv_LWrn)
      { S7_GenerateENO := "TRUE" } Move(in := "dbtags_Sterowanie".SetupControlPompownia.r_Pv_Hlm, out1 => "PID_Compact_1".sPid_Cmpt.r_Pv_Hlm)
      { S7_GenerateENO := "TRUE" } Move(in := "dbtags_Sterowanie".SetupControlPompownia.r_Pv_Llm, out1 => "PID_Compact_1".sPid_Cmpt.r_Pv_Llm)
   END_RUNG
   // the same network as SCL:
   // ENO of a box is taken as its EN; it also drops when the box reports an error
   "PID_Compact_1".sPid_Cmpt.r_Pv_HWrn := "dbtags_Sterowanie".SetupControlPompownia.r_Pv_HWrn;
   "PID_Compact_1".sPid_Cmpt.r_Pv_LWrn := "dbtags_Sterowanie".SetupControlPompownia.r_Pv_LWrn;
   "PID_Compact_1".sPid_Cmpt.r_Pv_Hlm := "dbtags_Sterowanie".SetupControlPompownia.r_Pv_Hlm;
   "PID_Compact_1".sPid_Cmpt.r_Pv_Llm := "dbtags_Sterowanie".SetupControlPompownia.r_Pv_Llm;
END_REGION

REGION Network 14: Zasuwa Z11 Tryb Automat
   RUNG wire#powerrail
      Move(in := 35980, out1 => "dbHoldRegSlave_to_MT101".instvValveZ11)
   END_RUNG
   // the same network as SCL:
   "dbHoldRegSlave_to_MT101".instvValveZ11 := 35980;
END_REGION

REGION Network 15: Zasuwa Z12 Tryb Automat
   RUNG wire#powerrail
      Move(in := 35980, out1 => "dbHoldRegSlave_to_MT101".instvValveZ12)
   END_RUNG
   // the same network as SCL:
   "dbHoldRegSlave_to_MT101".instvValveZ12 := 35980;
END_REGION

REGION Network 17: Inicjacja Inverter i zasilanie RS
   // Ustawienie gotowości po restarcie sterownika
   // Ustawienie przełacznika tryb pracy na Aut
   RUNG wire#powerrail
      Contact( "FirstScan" )
      wire#w1
      R_Coil( "dbzarządzanie".awaria_falownika_F1 )
   END_RUNG
   RUNG wire#w1
      R_Coil( "dbzarządzanie".awaria_falownika_F2 )
   END_RUNG
   RUNG wire#w1
      R_Coil( "dbzarządzanie".brak_zasilania_RS )
   END_RUNG
   RUNG wire#w1
      S_Coil( "dbzarządzanie".sterowanie_1.tryb_automat )
   END_RUNG
   // the same network as SCL:
   IF "FirstScan" THEN
       "dbzarządzanie".awaria_falownika_F1 := FALSE;
       "dbzarządzanie".awaria_falownika_F2 := FALSE;
       "dbzarządzanie".brak_zasilania_RS := FALSE;
       "dbzarządzanie".sterowanie_1.tryb_automat := TRUE;
   END_IF;
END_REGION

REGION Network 18: Startegia sterowania "Pompowna" , "Zbiorniki"
   // 0- wyłaczone, 1- dosilanie, 2- przetłaczanie, 3- automat,  4- ręczne
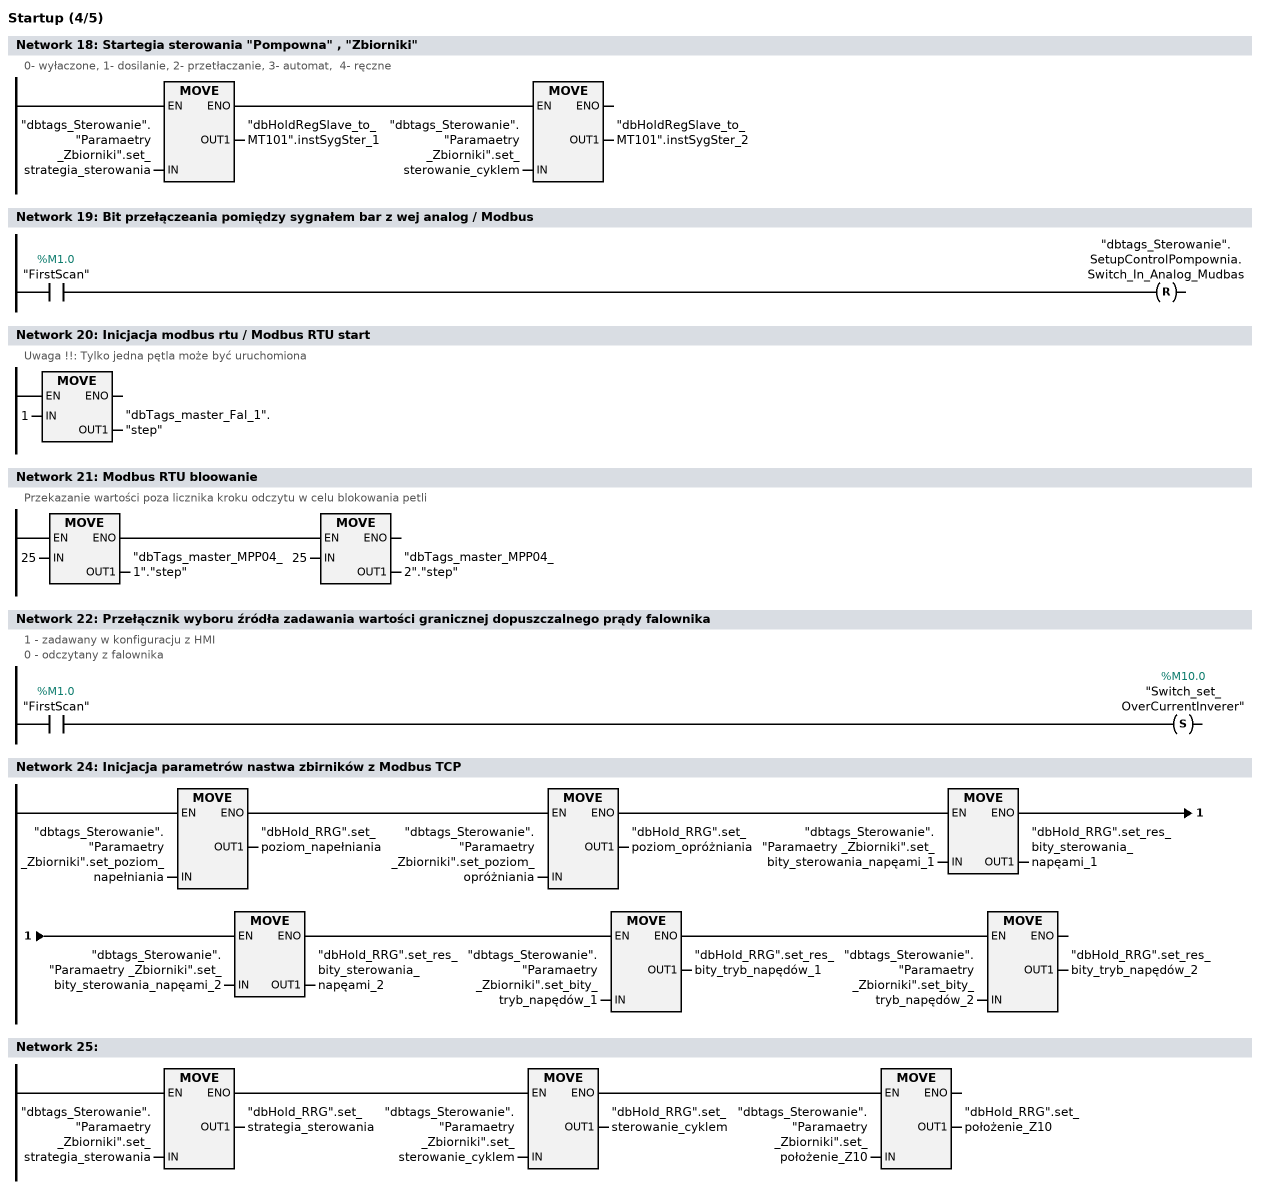
   RUNG wire#powerrail
      Move(in := "dbtags_Sterowanie"."Paramaetry _Zbiorniki".set_strategia_sterowania, out1 => "dbHoldRegSlave_to_MT101".instSygSter_1)
      Move(in := "dbtags_Sterowanie"."Paramaetry _Zbiorniki".set_sterowanie_cyklem, out1 => "dbHoldRegSlave_to_MT101".instSygSter_2)
   END_RUNG
   // the same network as SCL:
   "dbHoldRegSlave_to_MT101".instSygSter_1 := "dbtags_Sterowanie"."Paramaetry _Zbiorniki".set_strategia_sterowania;
   "dbHoldRegSlave_to_MT101".instSygSter_2 := "dbtags_Sterowanie"."Paramaetry _Zbiorniki".set_sterowanie_cyklem;
END_REGION

REGION Network 19: Bit przełączeania pomiędzy sygnałem bar z wej analog / Modbus
   RUNG wire#powerrail
      Contact( "FirstScan" )
      R_Coil( "dbtags_Sterowanie".SetupControlPompownia.Switch_In_Analog_Mudbas )
   END_RUNG
   // the same network as SCL:
   IF "FirstScan" THEN "dbtags_Sterowanie".SetupControlPompownia.Switch_In_Analog_Mudbas := FALSE; END_IF;
END_REGION

REGION Network 20: Inicjacja modbus rtu / Modbus RTU start
   // Uwaga !!: Tylko jedna pętla może być uruchomiona
   RUNG wire#powerrail
      { S7_GenerateENO := "TRUE" } Move(in := 1, out1 => "dbTags_master_Fal_1"."step")
   END_RUNG
   // the same network as SCL:
   "dbTags_master_Fal_1"."step" := 1;
END_REGION

REGION Network 21: Modbus RTU bloowanie
   // Przekazanie wartości poza licznika kroku odczytu w celu blokowania petli
   RUNG wire#powerrail
      { S7_GenerateENO := "TRUE" } Move(in := 25, out1 => "dbTags_master_MPP04_1"."step")
      { S7_GenerateENO := "TRUE" } Move(in := 25, out1 => "dbTags_master_MPP04_2"."step")
   END_RUNG
   // the same network as SCL:
   // ENO of a box is taken as its EN; it also drops when the box reports an error
   "dbTags_master_MPP04_1"."step" := 25;
   "dbTags_master_MPP04_2"."step" := 25;
END_REGION

REGION Network 22: Przełącznik wyboru źródła zadawania wartości granicznej dopuszczalnego prądy falownika
   // 1 - zadawany w konfiguracju z HMI
   // 0 - odczytany z falownika
   RUNG wire#powerrail
      Contact( "FirstScan" )
      S_Coil( "Switch_set_OverCurrentInverer" )
   END_RUNG
   // the same network as SCL:
   IF "FirstScan" THEN "Switch_set_OverCurrentInverer" := TRUE; END_IF;
END_REGION

REGION Network 23 (SCL): Ustawienie Setpoint SV do regulatora
   // Wartość ciśnienia zadanego zależna od wybranej strategii
   CASE "dbHoldRegSlave_to_MT101".instSygSter_1 OF
     1:
       "dbdane".Setpoint_SV := "dbtags_Sterowanie".SetupControlPompownia.set_barDN500_B5 ;
     2:
       "dbdane".Setpoint_SV := "dbtags_Sterowanie".SetupControlPompownia.set_barDN225_B6;
     3:
       "dbdane".Setpoint_SV := "dbdane".Setpoint_bar_automat ;

     ELSE
       "dbdane".Setpoint_SV := 0.0;
       ;
   END_CASE;
END_REGION

